	(*Allow Robots to Proceed Into Tool*)
	(*!!!!!This is the final OK to allow Robots Into the Tool Area, So it Better Be Ready!!!!!!!*)
	IF Enable_Motion
		THEN
			IF Load_Robots_Proceed1 AND Load_Robots_WorkingOK1 AND Load_Robots_Clear2 AND Seal_Robots_Clear AND Stud_Robots_Clear AND Turntable_Clear AND Weld_Robots_Clear AND Unload_Robots_Clear
				THEN Robots_Clear_ToProceed:=TRUE;
			ELSIF Load_Robots_Proceed2 AND Load_Robots_WorkingOK2 AND Load_Robots_Clear1 AND Seal_Robots_Clear AND Stud_Robots_Clear AND Turntable_Clear AND Weld_Robots_Clear AND Unload_Robots_Clear
				THEN Robots_Clear_ToProceed:=TRUE;
			ELSIF Seal_Robots_Proceed AND Seal_Robots_WorkingOK AND Load_Robots_Clear AND Stud_Robots_Clear AND Turntable_Clear AND Weld_Robots_Clear AND Unload_Robots_Clear
				THEN Robots_Clear_ToProceed:=TRUE;
			ELSIF Stud_Robots_Proceed AND Stud_Robots_WorkingOK AND Load_Robots_Clear AND Seal_Robots_Clear AND Turntable_Clear AND Weld_Robots_Clear AND Unload_Robots_Clear
				THEN Robots_Clear_ToProceed:=TRUE;
			ELSIF Weld_Robots_Proceed AND Weld_Robots_WorkingOK AND Load_Robots_Clear AND Seal_Robots_Clear AND Stud_Robots_Clear AND Turntable_Clear AND Unload_Robots_Clear
				THEN Robots_Clear_ToProceed:=TRUE;
			ELSIF Unload_Robots_Proceed1 AND Unload_Robots_WorkingOK1 AND Load_Robots_Clear AND Seal_Robots_Clear AND Stud_Robots_Clear AND Turntable_Clear AND Weld_Robots_Clear AND Unload_Robots_Clear2
				THEN Robots_Clear_ToProceed:=TRUE;
			ELSIF Unload_Robots_Proceed2 AND Unload_Robots_WorkingOK2 AND Load_Robots_Clear AND Seal_Robots_Clear AND Stud_Robots_Clear AND Turntable_Clear AND Weld_Robots_Clear AND Unload_Robots_Clear1
				THEN Robots_Clear_ToProceed:=TRUE;
			ELSE Robots_Clear_ToProceed:= FALSE;
			END_IF;
		ELSE Robots_Clear_ToProceed:= FALSE;
	END_IF;

(*+++++++++++++++++++++++++++++++++++++++++++++++ Task Complete Acks ++++++++++++++++++++++++++*)
	(*1st Load Complete Ack*)
	Load_Complete1_Ack:= Load_Robots_Complete1 AND Load_Complete1;

	(*2nd Load Complete Ack*)
	Load_Complete2_Ack:= Load_Robots_Complete2 AND Load_Complete2;

	(*Seal Complete Ack*)
	Seal_Complete_Ack:= Seal_Robots_Complete AND Sealing_Complete;

	(*Stud Complete Ack*)
	Stud_Complete_Ack:= Stud_Robots_Complete AND Stud_Complete;

	(*Sweep Complete ACK*)
	TurnA_Complete_Ack := TurntableA_Complete AND TurntableA_At_Robot;
	TurnB_Complete_Ack := TurntableB_Complete AND TurntableB_At_Robot;

	(*Weld Complete Ack*)
	Weld_Complete_Ack:= Weld_Robots_Complete AND Welding_Complete;

	(*Unload Complete Ack*)
	Unload_Complete1_Ack:= Unload_Robots_Complete1 AND Unload_Complete;

	(*Unload Complete Ack*)
	Unload_Complete2_Ack:= Unload_Robots_Complete2 AND Unload_Complete;






(*end*)
END_ACTION

ACTION Status_and_Faults:



(*^^^^^^^^^^^^^^^^^^^^^^^^^^^^^^^^^^^^^^ General Visualization ^^^^^^^^^^^^^^^^^^^^^^^^^^^^^^^^^^^^*)
	(*For Ready to Load Indicators*)
		(*Flash when tool should be loaded but load is not complete*)
		IF In_Auto AND Tool_At_Home AND NOT Welding_Complete AND All_Robots_Clear AND NOT All_Sensors_On.2
			THEN
				Ready_To_Load:= Pulse_500mS;
				(*Go solid when tool has been loaded properly*)
				(*Go solid when tool is ready to be unloaded*)
		ELSIF In_Auto AND All_Robots_Clear  AND ((Tool_At_Home AND NOT Welding_Complete AND All_Sensors_On.2 AND NOT Enable_Motion)
			OR (Tool_At_Unload.0 AND Welding_Complete AND (Sealing_Complete OR Sealer_Bypass) AND (Stud_Complete OR Stud_Bypass) AND TurntableA_At_Robot AND NOT All_Sensors_Off))
			THEN
				Ready_To_Load:= TRUE;
		ELSE
				Ready_To_Load:= FALSE;
		END_IF;
	(*For Red Stack Light Indicators*)
		Red_Lamp_Req:= PPFaults<>0 OR CLFaulted.0 OR CLFaulted.4 OR (NOT Sealer_Bypass AND MAIN.SL01.Disp1_Volume_NotOK AND (MAIN.R1.Task_ID_Ack=Seal_Fix01)) OR Load_Seq01.Faulted;


	(*Status Banners*)
		(*1 - Check Parts On Sub Check*)
		IF In_Auto AND NOT In_Manual AND NOT Cycle_Complete AND Tool_At_Load.0
			AND NOT Start_Load_Robots1 AND NOT Start_Load_Robots2 AND NOT Start_Seal_Robots AND NOT Start_Stud_Robots AND NOT Start_TurntableA
			AND NOT Start_TurntableB AND NOT Start_Weld_Robots AND NOT Start_Unload_Robots1 AND NOT Start_Unload_Robots2
			THEN
				IF NOT Dry_Cycle AND NOT All_Sensors_On.0
					THEN Status:= 1;
				ELSIF Dry_Cycle AND NOT Load_Complete1
					THEN Status:=1;
				END_IF;
		END_IF;
		(*2 - Sub Check OK*)
		IF In_Auto AND NOT In_Manual AND NOT Cycle_Complete AND Tool_At_Load.1
			AND NOT Start_Load_Robots1 AND NOT Start_Load_Robots2 AND NOT Start_Seal_Robots AND NOT Start_Stud_Robots AND NOT Start_TurntableA
			AND NOT Start_TurntableB AND NOT Start_Weld_Robots AND NOT Start_Unload_Robots1 AND NOT Start_Unload_Robots2
			THEN
				IF NOT Dry_Cycle AND NOT All_Sensors_On.1
					THEN Status:= 2;
				ELSIF Dry_Cycle AND NOT Load_Complete2
					THEN Status:=2;
				END_IF;
		END_IF;
		(*3 - Load Main Part*)
		IF In_Auto AND NOT In_Manual AND NOT Cycle_Complete AND Tool_At_Home
			AND NOT Start_Load_Robots1 AND NOT Start_Load_Robots2 AND NOT Start_Seal_Robots AND NOT Start_Stud_Robots AND NOT Start_TurntableA
			AND NOT Start_TurntableB AND NOT Start_Weld_Robots AND NOT Start_Unload_Robots1 AND NOT Start_Unload_Robots2
			THEN
				IF NOT Dry_Cycle AND NOT All_Sensors_On.2
					THEN Status:= 3;
				ELSIF Dry_Cycle AND NOT Load_Complete
					THEN Status:=3;
				END_IF;
		END_IF;
		(*10 - Load Parts Onto Tool*)
		IF In_Auto AND NOT In_Manual AND NOT Cycle_Complete AND Tool_At_Load.0
			AND NOT Start_Load_Robots1 AND NOT Start_Load_Robots2 AND NOT Start_Seal_Robots AND NOT Start_Stud_Robots AND NOT Start_TurntableA
			AND NOT Start_TurntableB AND NOT Start_Weld_Robots AND NOT Start_Unload_Robots1 AND NOT Start_Unload_Robots2
			THEN
				IF NOT Dry_Cycle AND NOT All_Sensors_On.2
					THEN Status:= 10;
				ELSIF Dry_Cycle AND NOT Load_Complete
					THEN Status:=10;
				END_IF;
		END_IF;
		(*11 - Robot(s) Loading*)
		IF ((Start_Load_Robots1 OR  Load_Robots_WorkingOK1) OR (Start_Load_Robots2 OR  Load_Robots_WorkingOK2)) AND In_Auto AND NOT In_Manual
			AND NOT Start_Seal_Robots AND NOT Start_Stud_Robots AND NOT Start_TurntableA
			AND NOT Start_TurntableB AND NOT Start_Weld_Robots AND NOT Start_Unload_Robots1 AND NOT Start_Unload_Robots2
			THEN Status:= 11;
		END_IF;
		(*12 - Parts Loaded OK*)
		IF In_Auto AND NOT In_Manual AND NOT Cycle_Complete
			AND NOT Start_Load_Robots1 AND NOT Start_Load_Robots2 AND NOT Start_Seal_Robots AND NOT Start_Stud_Robots AND NOT Start_TurntableA
			 AND NOT Start_TurntableB AND NOT Start_Weld_Robots AND NOT Start_Unload_Robots1 AND NOT Start_Unload_Robots2
			THEN
				IF (All_Sensors_On.2 AND Tool_At_Load.0) AND NOT Dry_Cycle
					THEN Status:= 12;
				ELSIF Load_Complete
					THEN Status:= 12;
				END_IF;
		END_IF;
		(*19 - Robot(s) Stud*)
		IF (Start_Stud_Robots OR Stud_Robots_WorkingOK) AND In_Auto AND NOT In_Manual
			AND NOT Start_Load_Robots1 AND NOT Start_Load_Robots2 AND NOT Start_Weld_Robots AND NOT Start_Seal_Robots AND NOT Start_TurntableA
			 AND NOT Start_TurntableB AND NOT Start_Unload_Robots1 AND NOT Start_Unload_Robots2
			THEN Status:= 19;
		END_IF;
		(*20 - Robot(s) Sealing*)
		IF (Start_Seal_Robots OR Seal_Robots_WorkingOK) AND In_Auto AND NOT In_Manual
			AND NOT Start_Load_Robots1 AND NOT Start_Load_Robots2 AND NOT Start_Weld_Robots AND NOT Start_Stud_Robots AND NOT Start_TurntableA
			 AND NOT Start_TurntableB AND NOT Start_Unload_Robots1 AND NOT Start_Unload_Robots2
			THEN Status:= 20;
		END_IF;
		(*21 - Robot(s) Welding*)
		IF (Start_Weld_Robots OR Weld_Robots_WorkingOK) AND In_Auto AND NOT In_Manual
			AND NOT Start_Load_Robots1 AND NOT Start_Load_Robots2 AND NOT Start_Seal_Robots AND NOT Start_Stud_Robots AND NOT Start_TurntableA
			 AND NOT Start_TurntableB AND NOT Start_Unload_Robots1 AND NOT Start_Unload_Robots2
			THEN Status:= 21;
		END_IF;
		(*22 - Welding Complete / Ready for Unload*)
		IF In_Auto AND NOT In_Manual AND NOT Cycle_Complete AND Welding_Complete
			AND NOT Start_Load_Robots1 AND NOT Start_Load_Robots2 AND NOT Start_Seal_Robots AND NOT Start_Stud_Robots AND NOT Start_TurntableA
			AND NOT Start_TurntableB AND NOT Start_Weld_Robots AND NOT Start_Unload_Robots1 AND NOT Start_Unload_Robots2
			THEN Status:= 22;
		END_IF;
		(*26 - Ready for Rotate*)
		IF (Start_TurntableA OR Start_TurntableB) AND In_Auto AND NOT In_Manual
			AND NOT Start_Load_Robots1 AND NOT Start_Load_Robots2 AND NOT Start_Seal_Robots AND NOT Start_Stud_Robots
			AND NOT Start_Weld_Robots AND NOT Start_Unload_Robots1 AND NOT Start_Unload_Robots2
			THEN Status := 26;
		END_IF;
		(*31 - Robot(s) Unloading*)
		IF (Start_Unload_Robots1 OR Unload_Robots_WorkingOK1 OR Start_Unload_Robots2 OR Unload_Robots_WorkingOK2) AND In_Auto AND NOT In_Manual
			AND NOT Start_Load_Robots1 AND NOT Start_Load_Robots2 AND NOT Start_Seal_Robots AND NOT Start_Stud_Robots AND NOT Start_TurntableA
			AND NOT Start_TurntableB AND NOT Start_Weld_Robots
			THEN Status:= 31;
		END_IF;
		(*32 - Unload Complete*)
		IF In_Auto AND NOT In_Manual AND NOT Cycle_Complete AND Unload_Complete
			AND NOT Start_Load_Robots1 AND NOT Start_Load_Robots2 AND NOT Start_Seal_Robots AND NOT Start_Stud_Robots AND NOT Start_TurntableA
			AND NOT Start_TurntableB AND NOT Start_Weld_Robots AND NOT Start_Unload_Robots1 AND NOT Start_Unload_Robots2
			THEN Status:= 32;
		END_IF;
		(*42 - Cycle Complete*)
		IF In_Auto AND NOT In_Manual AND Cycle_Complete AND All_Sensors_Off
			THEN Status:= 42;
		END_IF;
		(*50 - In Manual*)
		IF In_Manual
			THEN Status:= 50;
		END_IF;
		(*51 - Clamp Fault*)
		IF (CLFaults1>0 OR CLFaults2>0 OR CLFaults3>0 OR CLFaults4>0) AND In_Auto AND NOT In_Manual
			THEN Status:= 51;
		END_IF;
		(*52 - Part Present Sensor Fault*)
		IF PPFaults>0 AND In_Auto AND NOT In_Manual
			THEN Status:= 52;
		END_IF;
		(*53 - Nut Checks Failed Call QA*)
		IF QAChecks_Failed AND In_Auto AND NOT In_Manual
			THEN Status:= 53;
		END_IF;
		(*54 - Sealer Failed Call QA*)
		IF NOT Sealer_Bypass AND (MAIN.SL01.Disp1_Volume_NotOK AND (MAIN.R1.Task_ID_Ack=Seal_Fix01)) AND In_Auto AND NOT In_Manual
			THEN Status:= 54;
		END_IF;
		(*55 - Load Sequence Fault Call QA*)
		IF Load_Seq01.Faulted AND In_Auto AND NOT In_Manual
			THEN Status:= 55;
		END_IF;



(*$$$$$$$$$$$$$$$$$$$$$$$$$$$$$$$$$$$$$$$$$$$$$$$$$$$ Faults $$$$$$$$$$$$$$$$$$$$$$$$$$$$$$$$$$$$$$$$$$$$$$$$$$$$$$$*)

	(*Clamp/Cylider Faults Group 1*)
		IF CLFaults1>0
			THEN CLFaulted.1:=TRUE;
		ELSE
			CLFaulted.1:=FALSE;
		END_IF;
	(*Clamp/Cylider Faults Group 2*)
		IF CLFaults2>0
			THEN CLFaulted.2:=TRUE;
		ELSE
			CLFaulted.2:=FALSE;
		END_IF;
	(*Clamp/Cylider Faults Group 3*)
		IF CLFaults3>0
			THEN CLFaulted.3:=TRUE;
		ELSE
			CLFaulted.3:=FALSE;
		END_IF;
	(*Clamp/Cylinder Faults Group 4 - Reserved Flag for QA Check Motion Faults*)
		IF CLFaults4>0
			THEN CLFaulted.4:=TRUE;
		ELSE
			CLFaulted.4:=FALSE;
		END_IF;
	(*Bit 0 is designated as ANY Clamp Group Faulted*)
	IF CLFaulted.1 OR CLFaulted.2 OR CLFaulted.3
		THEN CLFaulted.0:= TRUE;
	ELSE CLFaulted.0 := FALSE;
	END_IF;

	(*Part Present Sensor Faults*)
		IF (PPFaults>0) OR (PPFaults1>0) OR (PPFaults2>0)
			THEN PPFaulted.0:=TRUE;
		ELSE
			PPFaulted.0:=FALSE;
		END_IF;
























(*end*)
END_ACTION

ACTION Task_Fix_Model_IDs:


	(*Develop Task IDs - See Global Variable, "TaskID_Record"*)

	IF (Start_Load_Robots1 OR Start_Load_Robots2) AND Enable_Motion
		THEN Task_ID:= Dropoff_Fix04;
	ELSIF Start_Seal_Robots AND Enable_Motion
		THEN Task_ID:= Seal_Fix04;
	ELSIF Start_Stud_Robots AND Enable_Motion
		THEN Task_ID:= Stud_Fix04;
	ELSIF Start_Weld_Robots AND Enable_Motion
		THEN Task_ID:= Weld_Fix04;
	ELSIF Start_TurnTableB AND Enable_Motion
		THEN Task_ID:= Sweep_Fix04;
	ELSIF (Start_Unload_Robots1 OR Start_Unload_Robots2) AND Enable_Motion
		THEN Task_ID:= Pickup_Fix04;
	ELSE Task_ID:= 0;
	END_IF;

	(*Develop Fixture ID*)
	Fix_ID:= N00.ID;					(*In Future Map Beckhoff Dip Switch Data From IP67 Block to Here*)

	(*Develop Model ID*)
	Model_ID:= Discrete_In.ModelData;
END_ACTION

ACTION Tool_States:


(*+++++++++++THIS AREA IS CUSTOM PER INSTALLATION AND WILL HAVE TO BE MODIFIED PER +++++++++++++*)
(*+++++++++++THIS AREA IS CUSTOM PER INSTALLATION AND WILL HAVE TO BE MODIFIED PER +++++++++++++*)

(*
						 MODEL ID MAP
					 -------------------
				Model ID :  Part ID  :   Tooling ID
					1  	 : 	 504     :     42
					2	 :   524     :	   42
					3	 :   543     :	   47
					4	 :   526     :	   46
					5	 :   536     :	   45
					6	 :   550     :	   44
					7	 :   571     :	   43
	
*)
	

	(*Tooling Position at HOME*)
	Tool_At_HOME:= 
				(((Model_ID=1) OR (Model_ID>3 OR (Model_ID=0)))		(*Model 504, 526, 536, 550, 571*)
				AND Clamp1RETD AND Clamp2RETD AND Clamp3RETD AND Clamp4RETD
				AND Clamp5RETD AND Clamp6RETD AND Clamp7RETD AND Clamp8RETD
				AND Clamp9RETD AND Clamp10RETD AND Clamp11RETD AND Clamp12RETD
				AND Clamp13RETD AND Clamp14RETD AND Clamp15RETD AND Clamp16RETD
				AND Clamp17RETD AND Clamp18RETD AND Clamp19RETD AND Clamp20RETD
				AND Clamp21RETD AND Clamp22RETD AND Pin1ADVD AND Pin2ADVD AND Pin3ADVD AND Pin4ADVD 
				AND Pin5RETD AND Pin6RETD AND Pin7ADVD AND Pin8ADVD AND Pin9ADVD AND Pin10ADVD 
				AND Pin11ADVD AND Pin12ADVD AND Pin13ADVD AND Pin14RETD AND Pin15RETD AND Pin16ADVD AND Pin17ADVD 
				AND Pin18ADVD AND Slide1ADVD AND Slide2ADVD AND Slide3RETD AND Slide4RETD AND Slide5RETD AND Slide6RETD
				AND Slide7RETD AND Slide8RETD AND Slide9RETD AND Slide10ADVD AND Slide11RETD AND Slide12RETD
				AND Slide13ADVD AND Slide14ADVD AND Swing1RETD AND Swing2RETD AND Swing3RETD)
			OR
				((Model_ID=2)		(*524*)
				AND Clamp1RETD AND Clamp2RETD AND Clamp3RETD AND Clamp4RETD
				AND Clamp5RETD AND Clamp6RETD AND Clamp7RETD AND Clamp8RETD
				AND Clamp9RETD AND Clamp10RETD AND Clamp11RETD AND Clamp12RETD
				AND Clamp13RETD AND Clamp14RETD AND Clamp15RETD AND Clamp16RETD
				AND Clamp17RETD AND Clamp18RETD AND Clamp19RETD AND Clamp20RETD
				AND Clamp21RETD AND Clamp22RETD AND Pin1ADVD AND Pin2ADVD AND Pin3ADVD AND Pin4ADVD 
				AND Pin5ADVD AND Pin6RETD AND Pin7ADVD AND Pin8ADVD AND Pin9ADVD AND Pin10ADVD 
				AND Pin11ADVD AND Pin12ADVD AND Pin13ADVD AND Pin14RETD AND Pin15ADVD AND Pin16ADVD AND Pin17ADVD 
				AND Pin18ADVD AND Slide1ADVD AND Slide2ADVD AND Slide3RETD AND Slide4RETD AND Slide5RETD AND Slide6RETD
				AND Slide7RETD AND Slide8RETD AND Slide9RETD AND Slide10ADVD AND Slide11RETD AND Slide12RETD
				AND Slide13ADVD AND Slide14ADVD AND Swing1RETD AND Swing2RETD AND Swing3RETD)
			OR
				((Model_ID=3)		(*543*)
				AND Clamp1RETD AND Clamp2RETD AND Clamp3RETD AND Clamp4RETD
				AND Clamp5RETD AND Clamp6RETD AND Clamp7RETD AND Clamp8RETD
				AND Clamp9RETD AND Clamp10RETD AND Clamp11RETD AND Clamp12RETD
				AND Clamp13RETD AND Clamp14RETD AND Clamp15RETD AND Clamp16RETD
				AND Clamp17RETD AND Clamp18RETD AND Clamp19RETD AND Clamp20RETD
				AND Clamp21RETD AND Clamp22RETD AND Pin1ADVD AND Pin2ADVD AND Pin3ADVD AND Pin4ADVD 
				AND Pin5RETD AND Pin6ADVD AND Pin7ADVD AND Pin8ADVD AND Pin9ADVD AND Pin10ADVD 
				AND Pin11ADVD AND Pin12ADVD AND Pin13ADVD AND Pin14ADVD AND Pin15RETD AND Pin16ADVD AND Pin17ADVD 
				AND Pin18ADVD AND Slide1ADVD AND Slide2ADVD AND Slide3RETD AND Slide4RETD AND Slide5RETD AND Slide6RETD
				AND Slide7RETD AND Slide8RETD AND Slide9RETD AND Slide10ADVD AND Slide11RETD AND Slide12RETD
				AND Slide13ADVD AND Slide14ADVD AND Swing1RETD AND Swing2RETD AND Swing3RETD);

	(*Tooling position to load parts*)
	Tool_At_Load.0:=
				(((Model_ID=1) OR (Model_ID>3))		(*Model 504, 526, 536, 550, 571*)
				AND Clamp1RETD AND Clamp2RETD AND Clamp3RETD AND Clamp4RETD
				AND Clamp5RETD AND Clamp6RETD AND Clamp7RETD AND Clamp8RETD
				AND Clamp9RETD AND Clamp10RETD AND Clamp11RETD AND Clamp12RETD
				AND Clamp13RETD AND Clamp14RETD AND Clamp15RETD AND Clamp16RETD
				AND Clamp17RETD AND Clamp18RETD AND Clamp19RETD AND Clamp20RETD
				AND Clamp21RETD AND Clamp22RETD AND Pin1ADVD AND Pin2ADVD AND Pin3ADVD AND Pin4ADVD 
				AND Pin5RETD AND Pin6RETD AND Pin7ADVD AND Pin8ADVD AND Pin9ADVD AND Pin10ADVD 
				AND Pin11ADVD AND Pin12ADVD AND Pin13ADVD AND Pin14RETD AND Pin15RETD AND Pin16ADVD AND Pin17ADVD 
				AND Pin18ADVD AND Slide1ADVD AND Slide2ADVD AND Slide3RETD AND Slide4RETD AND Slide5RETD AND Slide6RETD
				AND Slide7RETD AND Slide8RETD AND Slide9RETD AND Slide10ADVD AND Slide11RETD AND Slide12RETD
				AND Slide13ADVD AND Slide14ADVD AND Swing1RETD AND Swing2RETD AND Swing3RETD)
			OR
				((Model_ID=2)		(*Model 524*)
				AND Clamp1RETD AND Clamp2RETD AND Clamp3RETD AND Clamp4RETD
				AND Clamp5RETD AND Clamp6RETD AND Clamp7RETD AND Clamp8RETD
				AND Clamp9RETD AND Clamp10RETD AND Clamp11RETD AND Clamp12RETD
				AND Clamp13RETD AND Clamp14RETD AND Clamp15RETD AND Clamp16RETD
				AND Clamp17RETD AND Clamp18RETD AND Clamp19RETD AND Clamp20RETD
				AND Clamp21RETD AND Clamp22RETD AND Pin1ADVD AND Pin2ADVD AND Pin3ADVD AND Pin4ADVD 
				AND Pin5ADVD AND Pin6RETD AND Pin7ADVD AND Pin8ADVD AND Pin9ADVD AND Pin10ADVD 
				AND Pin11ADVD AND Pin12ADVD AND Pin13ADVD AND Pin14RETD AND Pin15ADVD AND Pin16ADVD AND Pin17ADVD 
				AND Pin18ADVD AND Slide1ADVD AND Slide2ADVD AND Slide3RETD AND Slide4RETD AND Slide5RETD AND Slide6RETD
				AND Slide7RETD AND Slide8RETD AND Slide9RETD AND Slide10ADVD AND Slide11RETD AND Slide12RETD
				AND Slide13ADVD AND Slide14ADVD AND Swing1RETD AND Swing2RETD AND Swing3RETD)
			OR
				((Model_ID=3)		(*Model 543*)
				AND Clamp1RETD AND Clamp2RETD AND Clamp3RETD AND Clamp4RETD
				AND Clamp5RETD AND Clamp6RETD AND Clamp7RETD AND Clamp8RETD
				AND Clamp9RETD AND Clamp10RETD AND Clamp11RETD AND Clamp12RETD
				AND Clamp13RETD AND Clamp14RETD AND Clamp15RETD AND Clamp16RETD
				AND Clamp17RETD AND Clamp18RETD AND Clamp19RETD AND Clamp20RETD
				AND Clamp21RETD AND Clamp22RETD AND Pin1ADVD AND Pin2ADVD AND Pin3ADVD AND Pin4ADVD 
				AND Pin5RETD AND Pin6ADVD AND Pin7ADVD AND Pin8ADVD AND Pin9ADVD AND Pin10ADVD 
				AND Pin11ADVD AND Pin12ADVD AND Pin13ADVD AND Pin14ADVD AND Pin15RETD AND Pin16ADVD AND Pin17ADVD 
				AND Pin18ADVD AND Slide1ADVD AND Slide2ADVD AND Slide3RETD AND Slide4RETD AND Slide5RETD AND Slide6RETD
				AND Slide7RETD AND Slide8RETD AND Slide9RETD AND Slide10ADVD AND Slide11RETD AND Slide12RETD
				AND Slide13ADVD AND Slide14ADVD AND Swing1RETD AND Swing2RETD AND Swing3RETD);
	
	(*Tooling position on Loading Complete*)	
	Tool_At_Load.1:= 
				(((Model_ID=1) OR (Model_ID>3))		(*Model 504, 526, 536, 550, 571*)
				AND Clamp1ADVD AND Clamp2ADVD AND Clamp3ADVD AND Clamp4ADVD AND Clamp5ADVD AND Clamp5ADVD AND Clamp5ADVD
				AND Clamp6ADVD AND Clamp7ADVD AND Clamp8ADVD AND Clamp9ADVD AND Clamp10ADVD AND Clamp11ADVD AND Clamp12ADVD
				AND Clamp13ADVD AND Clamp14ADVD AND Clamp15ADVD AND Clamp16ADVD AND Clamp17ADVD AND Clamp18ADVD AND Clamp19ADVD
				AND Clamp20ADVD AND Clamp21ADVD AND Clamp22ADVD AND Pin1ADVD AND Pin2ADVD AND Pin3ADVD AND Pin4ADVD AND Pin5RETD
				AND Pin6RETD AND Pin7ADVD AND Pin8ADVD AND Pin9ADVD AND Pin10ADVD AND Pin11ADVD AND Pin12ADVD AND Pin13ADVD
				AND Pin14RETD AND Pin15RETD AND Pin16ADVD AND Pin17ADVD AND Pin18ADVD AND Slide1ADVD AND Slide2ADVD AND Slide3ADVD
				AND Slide4ADVD AND Slide5ADVD AND Slide6ADVD AND Slide7ADVD AND Slide8ADVD AND Slide9ADVD AND Slide10ADVD AND Slide11ADVD
				AND Slide12ADVD AND Slide13ADVD AND Slide14ADVD AND Swing1ADVD AND Swing2ADVD AND Swing3ADVD)
			OR
				((Model_ID=2)		(*Model 524*)
				AND Clamp1ADVD AND Clamp2ADVD AND Clamp3ADVD AND Clamp4ADVD AND Clamp5ADVD AND Clamp5ADVD AND Clamp5ADVD
				AND Clamp6ADVD AND Clamp7ADVD AND Clamp8ADVD AND Clamp9ADVD AND Clamp10ADVD AND Clamp11ADVD AND Clamp12ADVD
				AND Clamp13ADVD AND Clamp14ADVD AND Clamp15ADVD AND Clamp16ADVD AND Clamp17ADVD AND Clamp18ADVD AND Clamp19ADVD
				AND Clamp20ADVD AND Clamp21ADVD AND Clamp22ADVD AND Pin1ADVD AND Pin2ADVD AND Pin3ADVD AND Pin4ADVD AND Pin5ADVD
				AND Pin6RETD AND Pin7ADVD AND Pin8ADVD AND Pin9ADVD AND Pin10ADVD AND Pin11ADVD AND Pin12ADVD AND Pin13ADVD
				AND Pin14RETD AND Pin15ADVD AND Pin16ADVD AND Pin17ADVD AND Pin18ADVD AND Slide1ADVD AND Slide2ADVD AND Slide3ADVD
				AND Slide4ADVD AND Slide5ADVD AND Slide6ADVD AND Slide7ADVD AND Slide8ADVD AND Slide9ADVD AND Slide10ADVD AND Slide11ADVD
				AND Slide12ADVD AND Slide13ADVD AND Slide14ADVD AND Swing1ADVD AND Swing2ADVD AND Swing3ADVD)
			OR
				((Model_ID=3)		(*Model 543*)
				AND Clamp1ADVD AND Clamp2ADVD AND Clamp3ADVD AND Clamp4ADVD AND Clamp5ADVD AND Clamp5ADVD AND Clamp5ADVD
				AND Clamp6ADVD AND Clamp7ADVD AND Clamp8ADVD AND Clamp9ADVD AND Clamp10ADVD AND Clamp11ADVD AND Clamp12ADVD
				AND Clamp13ADVD AND Clamp14ADVD AND Clamp15ADVD AND Clamp16ADVD AND Clamp17ADVD AND Clamp18ADVD AND Clamp19ADVD
				AND Clamp20ADVD AND Clamp21ADVD AND Clamp22ADVD AND Pin1ADVD AND Pin2ADVD AND Pin3ADVD AND Pin4ADVD AND Pin5RETD
				AND Pin6ADVD AND Pin7ADVD AND Pin8ADVD AND Pin9ADVD AND Pin10ADVD AND Pin11ADVD AND Pin12ADVD AND Pin13ADVD
				AND Pin14ADVD AND Pin15RETD AND Pin16ADVD AND Pin17ADVD AND Pin18ADVD AND Slide1ADVD AND Slide2ADVD AND Slide3ADVD
				AND Slide4ADVD AND Slide5ADVD AND Slide6ADVD AND Slide7ADVD AND Slide8ADVD AND Slide9ADVD AND Slide10ADVD AND Slide11ADVD
				AND Slide12ADVD AND Slide13ADVD AND Slide14ADVD AND Swing1ADVD AND Swing2ADVD AND Swing3ADVD);
	Tool_At_Load.2:= FALSE;
	Tool_At_Load.3:= FALSE;
	Tool_At_Load.4:= FALSE;


	Tool_At_Seal.0:= FALSE;
	Tool_At_Seal.1:= FALSE;
	Tool_At_Seal.2:= FALSE;
	Tool_At_Seal.3:= FALSE;
	Tool_At_Seal.4:= FALSE;


	Tool_At_Stud.0:= FALSE;
	Tool_At_Stud.1:= FALSE;
	Tool_At_Stud.2:= FALSE;
	Tool_At_Stud.3:= FALSE;
	Tool_At_Stud.4:= FALSE;

	(*Tooling position for ready to rotate*)
	Tool_At_Rotate.0:= 
				(((Model_ID=1) OR (Model_ID>3))		(*Model 504, 526, 536, 550, 571*)
				AND Clamp1ADVD AND Clamp2ADVD AND Clamp3ADVD AND Clamp4ADVD AND Clamp5ADVD AND Clamp5ADVD AND Clamp5ADVD
				AND Clamp6ADVD AND Clamp7ADVD AND Clamp8ADVD AND Clamp9ADVD AND Clamp10ADVD AND Clamp11ADVD AND Clamp12ADVD
				AND Clamp13ADVD AND Clamp14ADVD AND Clamp15ADVD AND Clamp16ADVD AND Clamp17ADVD AND Clamp18ADVD AND Clamp19ADVD
				AND Clamp20ADVD AND Clamp21ADVD AND Clamp22ADVD AND Pin1ADVD AND Pin2ADVD AND Pin3ADVD AND Pin4ADVD AND Pin5RETD
				AND Pin6RETD AND Pin7ADVD AND Pin8ADVD AND Pin9ADVD AND Pin10ADVD AND Pin11ADVD AND Pin12ADVD AND Pin13ADVD
				AND Pin14RETD AND Pin15RETD AND Pin16ADVD AND Pin17ADVD AND Pin18ADVD AND Slide1ADVD AND Slide2ADVD AND Slide3ADVD
				AND Slide4ADVD AND Slide5ADVD AND Slide6ADVD AND Slide7ADVD AND Slide8ADVD AND Slide9ADVD AND Slide10ADVD AND Slide11ADVD
				AND Slide12ADVD AND Slide13ADVD AND Slide14ADVD AND Swing1ADVD AND Swing2ADVD AND Swing3ADVD)
			OR
				((Model_ID=2)		(*Model 524*)
				AND Clamp1ADVD AND Clamp2ADVD AND Clamp3ADVD AND Clamp4ADVD AND Clamp5ADVD AND Clamp5ADVD AND Clamp5ADVD
				AND Clamp6ADVD AND Clamp7ADVD AND Clamp8ADVD AND Clamp9ADVD AND Clamp10ADVD AND Clamp11ADVD AND Clamp12ADVD
				AND Clamp13ADVD AND Clamp14ADVD AND Clamp15ADVD AND Clamp16ADVD AND Clamp17ADVD AND Clamp18ADVD AND Clamp19ADVD
				AND Clamp20ADVD AND Clamp21ADVD AND Clamp22ADVD AND Pin1ADVD AND Pin2ADVD AND Pin3ADVD AND Pin4ADVD AND Pin5ADVD
				AND Pin6RETD AND Pin7ADVD AND Pin8ADVD AND Pin9ADVD AND Pin10ADVD AND Pin11ADVD AND Pin12ADVD AND Pin13ADVD
				AND Pin14RETD AND Pin15ADVD AND Pin16ADVD AND Pin17ADVD AND Pin18ADVD AND Slide1ADVD AND Slide2ADVD AND Slide3ADVD
				AND Slide4ADVD AND Slide5ADVD AND Slide6ADVD AND Slide7ADVD AND Slide8ADVD AND Slide9ADVD AND Slide10ADVD AND Slide11ADVD
				AND Slide12ADVD AND Slide13ADVD AND Slide14ADVD AND Swing1ADVD AND Swing2ADVD AND Swing3ADVD)
			OR
				((Model_ID=3)		(*Model 543*)
				AND Clamp1ADVD AND Clamp2ADVD AND Clamp3ADVD AND Clamp4ADVD AND Clamp5ADVD AND Clamp5ADVD AND Clamp5ADVD
				AND Clamp6ADVD AND Clamp7ADVD AND Clamp8ADVD AND Clamp9ADVD AND Clamp10ADVD AND Clamp11ADVD AND Clamp12ADVD
				AND Clamp13ADVD AND Clamp14ADVD AND Clamp15ADVD AND Clamp16ADVD AND Clamp17ADVD AND Clamp18ADVD AND Clamp19ADVD
				AND Clamp20ADVD AND Clamp21ADVD AND Clamp22ADVD AND Pin1ADVD AND Pin2ADVD AND Pin3ADVD AND Pin4ADVD AND Pin5RETD
				AND Pin6ADVD AND Pin7ADVD AND Pin8ADVD AND Pin9ADVD AND Pin10ADVD AND Pin11ADVD AND Pin12ADVD AND Pin13ADVD
				AND Pin14ADVD AND Pin15RETD AND Pin16ADVD AND Pin17ADVD AND Pin18ADVD AND Slide1ADVD AND Slide2ADVD AND Slide3ADVD
				AND Slide4ADVD AND Slide5ADVD AND Slide6ADVD AND Slide7ADVD AND Slide8ADVD AND Slide9ADVD AND Slide10ADVD AND Slide11ADVD
				AND Slide12ADVD AND Slide13ADVD AND Slide14ADVD AND Swing1ADVD AND Swing2ADVD AND Swing3ADVD);
				
	Tool_At_Rotate.1:= FALSE;
	Tool_At_Rotate.2:= FALSE;
	Tool_At_Rotate.3:= FALSE;
	Tool_At_Rotate.4:= FALSE;

	(*Tooling position for welding*)
	Tool_At_Weld.0:= 
				(((Model_ID=1) OR (Model_ID>3))		(*Model 504, 526, 536, 550, 571*)
				AND Clamp1ADVD AND Clamp2ADVD AND Clamp3ADVD AND Clamp4ADVD AND Clamp5ADVD AND Clamp5ADVD AND Clamp5ADVD
				AND Clamp6ADVD AND Clamp7ADVD AND Clamp8ADVD AND Clamp9ADVD AND Clamp10ADVD AND Clamp11ADVD AND Clamp12ADVD
				AND Clamp13ADVD AND Clamp14ADVD AND Clamp15ADVD AND Clamp16ADVD AND Clamp17ADVD AND Clamp18ADVD AND Clamp19ADVD
				AND Clamp20ADVD AND Clamp21ADVD AND Clamp22ADVD AND Pin1ADVD AND Pin2ADVD AND Pin3ADVD AND Pin4ADVD AND Pin5RETD
				AND Pin6RETD AND Pin7ADVD AND Pin8ADVD AND Pin9ADVD AND Pin10ADVD AND Pin11ADVD AND Pin12ADVD AND Pin13ADVD
				AND Pin14RETD AND Pin15RETD AND Pin16ADVD AND Pin17ADVD AND Pin18ADVD AND Slide1ADVD AND Slide2ADVD AND Slide3ADVD
				AND Slide4ADVD AND Slide5ADVD AND Slide6ADVD AND Slide7ADVD AND Slide8ADVD AND Slide9ADVD AND Slide10ADVD AND Slide11ADVD
				AND Slide12ADVD AND Slide13ADVD AND Slide14ADVD AND Swing1ADVD AND Swing2ADVD AND Swing3ADVD)
			OR
				((Model_ID=2)		(*Model 524*)
				AND Clamp1ADVD AND Clamp2ADVD AND Clamp3ADVD AND Clamp4ADVD AND Clamp5ADVD AND Clamp5ADVD AND Clamp5ADVD
				AND Clamp6ADVD AND Clamp7ADVD AND Clamp8ADVD AND Clamp9ADVD AND Clamp10ADVD AND Clamp11ADVD AND Clamp12ADVD
				AND Clamp13ADVD AND Clamp14ADVD AND Clamp15ADVD AND Clamp16ADVD AND Clamp17ADVD AND Clamp18ADVD AND Clamp19ADVD
				AND Clamp20ADVD AND Clamp21ADVD AND Clamp22ADVD AND Pin1ADVD AND Pin2ADVD AND Pin3ADVD AND Pin4ADVD AND Pin5ADVD
				AND Pin6RETD AND Pin7ADVD AND Pin8ADVD AND Pin9ADVD AND Pin10ADVD AND Pin11ADVD AND Pin12ADVD AND Pin13ADVD
				AND Pin14RETD AND Pin15ADVD AND Pin16ADVD AND Pin17ADVD AND Pin18ADVD AND Slide1ADVD AND Slide2ADVD AND Slide3ADVD
				AND Slide4ADVD AND Slide5ADVD AND Slide6ADVD AND Slide7ADVD AND Slide8ADVD AND Slide9ADVD AND Slide10ADVD AND Slide11ADVD
				AND Slide12ADVD AND Slide13ADVD AND Slide14ADVD AND Swing1ADVD AND Swing2ADVD AND Swing3ADVD)
			OR
				((Model_ID=3)		(*Model 543*)
				AND Clamp1ADVD AND Clamp2ADVD AND Clamp3ADVD AND Clamp4ADVD AND Clamp5ADVD AND Clamp5ADVD AND Clamp5ADVD
				AND Clamp6ADVD AND Clamp7ADVD AND Clamp8ADVD AND Clamp9ADVD AND Clamp10ADVD AND Clamp11ADVD AND Clamp12ADVD
				AND Clamp13ADVD AND Clamp14ADVD AND Clamp15ADVD AND Clamp16ADVD AND Clamp17ADVD AND Clamp18ADVD AND Clamp19ADVD
				AND Clamp20ADVD AND Clamp21ADVD AND Clamp22ADVD AND Pin1ADVD AND Pin2ADVD AND Pin3ADVD AND Pin4ADVD AND Pin5RETD
				AND Pin6ADVD AND Pin7ADVD AND Pin8ADVD AND Pin9ADVD AND Pin10ADVD AND Pin11ADVD AND Pin12ADVD AND Pin13ADVD
				AND Pin14ADVD AND Pin15RETD AND Pin16ADVD AND Pin17ADVD AND Pin18ADVD AND Slide1ADVD AND Slide2ADVD AND Slide3ADVD
				AND Slide4ADVD AND Slide5ADVD AND Slide6ADVD AND Slide7ADVD AND Slide8ADVD AND Slide9ADVD AND Slide10ADVD AND Slide11ADVD
				AND Slide12ADVD AND Slide13ADVD AND Slide14ADVD AND Swing1ADVD AND Swing2ADVD AND Swing3ADVD);
	Tool_At_Weld.1:= FALSE;
	Tool_At_Weld.2:= FALSE;
	Tool_At_Weld.3:= FALSE;
	Tool_At_Weld.4:= FALSE;

	(*Tooling position for unload*)
	Tool_At_Unload.0:=Clamp1RETD AND Clamp2RETD AND Clamp3RETD AND Clamp4RETD
				AND Clamp5RETD AND Clamp6RETD AND Clamp7RETD AND Clamp8RETD
				AND Clamp9RETD AND Clamp10RETD AND Clamp11RETD AND Clamp12RETD
				AND Clamp13RETD AND Clamp14RETD AND Clamp15RETD AND Clamp16RETD
				AND Clamp17RETD AND Clamp18RETD AND Clamp19RETD AND Clamp20RETD
				AND Clamp21RETD AND Clamp22RETD AND Pin1RETD AND Pin2RETD AND Pin3RETD AND Pin4RETD AND Pin5RETD
				AND Pin6RETD AND Pin7RETD AND Pin8RETD AND Pin9RETD AND Pin10RETD AND Pin11RETD AND Pin12RETD 
				AND Pin13RETD AND Pin14RETD AND Pin15RETD AND Pin16RETD AND Pin17RETD AND Pin18RETD
				AND Slide1RETD AND Slide2RETD AND Slide3RETD AND Slide4RETD AND Slide5RETD AND Slide6RETD
				AND Slide7RETD AND Slide8RETD AND Slide9RETD AND Slide10RETD AND Slide11RETD AND Slide12RETD
				AND Slide13RETD AND Slide14RETD AND Swing1RETD AND Swing2RETD AND Swing3RETD;
	Tool_At_Unload.1:=FALSE;
	Tool_At_Unload.2:= FALSE;
	Tool_At_Unload.3:= FALSE;
	Tool_At_Unload.4:= FALSE;







































(*end*)
END_ACTION

ACTION Tool_VBSeq_Repos:
(*+++++++++++THIS AREA IS CUSTOM PER INSTALLATION AND WILL HAVE TO BE MODIFIED PER +++++++++++++*)
(*+++++++++++THIS AREA IS CUSTOM PER INSTALLATION AND WILL HAVE TO BE MODIFIED PER +++++++++++++*)


(*!!!!!!!!!!!!!!!!!!!!!!!!!!!!!!!!!!!!!!!!!! Tool Motion Control !!!!!!!!!!!!!!!!!!!!!!!!!!!!!!!*)

(*----------------------------------------- Clamp / Unclamp Steps -------------------------------*)

(*$$$$$$$$$$$$$$$$$$$$$$$$$$$$$$$$$$ Develop Clamp and Unclamp Interlocks $$$$$$$$$$$$$$$$$$$$$$*)
(* Note: This is one method to create valve bank commands for clamp and unclamp sequencing
you are welcome to use the direct method as well*)


	(*---------------------------------------------------------Start Clamp Sequence---------------------------------------------------------*)
	
	(*First Stage Clamping*)		(*V8, V10 ADV, IF Model 2 then V2 ADV, IF Model 3 then V5 ADV*)
	Clamp_Step.0:= Auto_Run AND NOT Welding_Complete OR (Cycle_Complete AND NOT Tool_At_Home AND All_Sensors_Off);
	
	
	(*Second Stage Clamping*)		(*V7, V9, V11 ADV, IF Model 2 then V1 ADV, IF Model 3 V4 ADV*)
	
	(*Model 504, 526, 536, 550, 571*)
	IF (Model_ID=1) OR (Model_ID>3) THEN		
				Clamp_Step.1:=  Clamp_Step.0 AND Load_Complete AND NOT Cycle_Complete AND
								(*V8*)
								(Pin1ADVD AND Pin2ADVD AND Pin3ADVD AND Pin4ADVD AND Pin7ADVD 
								AND Pin9ADVD AND Pin16ADVD AND Pin17ADVD AND Pin18ADVD AND Slide10ADVD)
								(*V10*)
								AND (Pin8ADVD AND Pin10ADVD AND Pin11ADVD AND Pin12ADVD AND Pin13ADVD 
								AND Slide1ADVD AND Slide2ADVD AND Slide13ADVD AND Slide14ADVD);
		(*Model 524*)						
		ELSIF (Model_ID=2) THEN					
				Clamp_Step.1:=  Clamp_Step.0 AND Load_Complete AND NOT Cycle_Complete AND 
								(*V2*)
								(Pin5ADVD AND Pin15ADVD)
								(*V8*)
								AND (Pin1ADVD AND Pin2ADVD AND Pin3ADVD AND Pin4ADVD AND Pin7ADVD 
								AND Pin9ADVD AND Pin16ADVD AND Pin17ADVD AND Pin18ADVD AND Slide10ADVD)
								(*V10*)
								AND (Pin8ADVD AND Pin10ADVD AND Pin11ADVD AND Pin12ADVD AND Pin13ADVD 
								AND Slide1ADVD AND Slide2ADVD AND Slide13ADVD AND Slide14ADVD);
		(*Model 543*)			
		ELSIF (Model_ID=3) THEN					
				Clamp_Step.1:=  Clamp_Step.0 AND Load_Complete AND NOT Cycle_Complete AND 
								(*V5*)
								(Pin6ADVD AND Pin14ADVD)
								(*V8*)
								AND (Pin1ADVD AND Pin2ADVD AND Pin3ADVD AND Pin4ADVD AND Pin7ADVD 
								AND Pin9ADVD AND Pin16ADVD AND Pin17ADVD AND Pin18ADVD AND Slide10ADVD)
								(*V10*)
								AND (Pin8ADVD AND Pin10ADVD AND Pin11ADVD AND Pin12ADVD AND Pin13ADVD 
								AND Slide1ADVD AND Slide2ADVD AND Slide13ADVD AND Slide14ADVD);						
	END_IF

	
	(*Third Stage Clamping*)		(*V13 ADV*)
	
	(*Model 504, 526, 536, 550, 571*)
	IF (Model_ID=1) OR (Model_ID>3) THEN
				Clamp_Step.2:= 	Clamp_Step.1 AND 
								(*V7*)
								(Clamp3ADVD AND Clamp18ADVD)
								(*V9*)
								AND (Clamp1ADVD AND Clamp2ADVD AND Clamp4ADVD AND Clamp5ADVD AND Clamp10ADVD 
								AND Clamp14ADVD AND Clamp21ADVD AND Clamp22ADVD)
								(*V11*)
								AND (Clamp9ADVD AND Clamp12ADVD AND Clamp13ADVD AND Clamp16ADVD);

		ELSIF (Model_ID=2) THEN
				Clamp_Step.2:= 	Clamp_Step.1 AND 
								(*V7*)
								(Clamp3ADVD AND Clamp18ADVD)
								(*V9*)
								AND (Clamp1ADVD AND Clamp2ADVD AND Clamp4ADVD AND Clamp5ADVD AND Clamp10ADVD 
								AND Clamp14ADVD AND Clamp21ADVD AND Clamp22ADVD)
								(*V11*)
								AND (Clamp9ADVD AND Clamp12ADVD AND Clamp13ADVD AND Clamp16ADVD)
								(*V1*)
								AND (Clamp6ADVD AND Clamp20ADVD);
		ELSIF (Model_ID=3) THEN
				Clamp_Step.2:= 	Clamp_Step.1 AND 
								(*V7*)
								(Clamp3ADVD AND Clamp18ADVD)
								(*V9*)
								AND (Clamp1ADVD AND Clamp2ADVD AND Clamp4ADVD AND Clamp5ADVD AND Clamp10ADVD 
								AND Clamp14ADVD AND Clamp21ADVD AND Clamp22ADVD)
								(*V11*)
								AND (Clamp9ADVD AND Clamp12ADVD AND Clamp13ADVD AND Clamp16ADVD)
								(*V4*)
								AND (Clamp8ADVD AND Clamp19ADVD);
	END_IF


	(*Forth Stage Clamping*)		(*V12 ADV, IF Model 2 V3 ADV, IF Model 3 V6 ADV*)
	
	Clamp_Step.3:= Clamp_Step.2 AND 
					(*V13*)
					(Clamp7ADVD AND Clamp11ADVD AND Clamp15ADVD AND Clamp17ADVD);




	(*---------------------------------------------------------Start Unclamp Sequence---------------------------------------------------------*)

	(*First Stage Unclamping*)		(*V7, V9, V11 RET, IF Model 2 V1 RET, IF Model 3 V4 RET*)

	Unclamp_Step.0:= (Welding_Complete AND TurnTableA_At_Robot);


	(*Second Stage Unclamping*)		(*V8, V10 RET, IF Model 2 V2 RET, IF Model 3 V5 RET*)
	(*Model 504, 526, 536, 550, 571*)
	IF (Model_ID=1) OR (Model_ID>3) THEN
			Unclamp_Step.1:= Unclamp_Step.0 AND 
								(*V7*)
								(Clamp3RETD AND Clamp18RETD)
								(*V9*)
								AND (Clamp1RETD AND Clamp2RETD AND Clamp4RETD AND Clamp5RETD AND Clamp10RETD AND Clamp14RETD AND Clamp21RETD AND Clamp22RETD)
								(*V11*)
								AND (Clamp9RETD AND Clamp12RETD AND Clamp13RETD AND Clamp16RETD);
		(*Model 524*)							
		ELSIF (Model_ID=2) THEN
				Unclamp_Step.1:= Unclamp_Step.0 AND 
									(*V7*)
									(Clamp3RETD AND Clamp18RETD)
									(*V9*)
									AND (Clamp1RETD AND Clamp2RETD AND Clamp4RETD AND Clamp5RETD AND Clamp10RETD AND Clamp14RETD AND Clamp21RETD AND Clamp22RETD)
									(*V11*)
									AND (Clamp9RETD AND Clamp12RETD AND Clamp13RETD AND Clamp16RETD)
									(*V1*)
									AND (Clamp6RETD AND Clamp20RETD);
		(*Model 543*)
		ELSIF (Model_ID=3) THEN							
				Unclamp_Step.1:= Unclamp_Step.0 AND 
									(*V7*)
									(Clamp3RETD AND Clamp18RETD)
									(*V9*)
									AND (Clamp1RETD AND Clamp2RETD AND Clamp4RETD AND Clamp5RETD AND Clamp10RETD AND Clamp14RETD AND Clamp21RETD AND Clamp22RETD)
									(*V11*)
									AND (Clamp9RETD AND Clamp12RETD AND Clamp13RETD AND Clamp16RETD)
									(*V4*)
									AND (Clamp8RETD AND Clamp19RETD);
	END_IF

	
	(*Third Stage Unclamping*)		(*V12 RET, IF Model 2 V3 RET, IF Model 3 V6 RET*)
	(*Model 504, 526, 536, 550, 571*)
	IF (Model_ID=1) OR (Model_ID>3) THEN
			Unclamp_Step.2:= Unclamp_Step.1 AND 
						(*V8*)
						(Pin1RETD AND Pin2RETD AND Pin3RETD AND Pin4RETD AND Pin7RETD AND Pin9RETD AND Pin16RETD AND Pin17RETD AND Pin18RETD AND Slide10RETD)
						(*V10*)
						AND (Pin8RETD AND Pin10RETD AND Pin11RETD AND Pin12RETD AND Pin13RETD AND Slide1RETD AND Slide2RETD AND Slide13RETD AND Slide14RETD);
		(*Model 524*)
		ELSIF (Model_ID=2) THEN
				Unclamp_Step.2:= Unclamp_Step.1 AND 
							(*V8*)
							(Pin1RETD AND Pin2RETD AND Pin3RETD AND Pin4RETD AND Pin7RETD AND Pin9RETD AND Pin16RETD AND Pin17RETD AND Pin18RETD AND Slide10RETD)
							(*V10*)
							AND (Pin8RETD AND Pin10RETD AND Pin11RETD AND Pin12RETD AND Pin13RETD AND Slide1RETD AND Slide2RETD AND Slide13RETD AND Slide14RETD)
							(*V2*)
							AND (Pin5RETD AND Pin15RETD);
		(*Model 543*)
		ELSIF (Model_ID=3) THEN
				Unclamp_Step.2:= Unclamp_Step.1 AND 
							(*V8*)
							(Pin1RETD AND Pin2RETD AND Pin3RETD AND Pin4RETD AND Pin7RETD AND Pin9RETD AND Pin16RETD AND Pin17RETD AND Pin18RETD AND Slide10RETD)
							(*V10*)
							AND (Pin8RETD AND Pin10RETD AND Pin11RETD AND Pin12RETD AND Pin13RETD AND Slide1RETD AND Slide2RETD AND Slide13RETD AND Slide14RETD)
							(*V5*)
							AND (Pin6RETD AND Pin14RETD);
	
	END_IF

	(*Fourth Stage Unclamping*)		(*V13 RET*)
	(*Model 504, 526, 536, 550, 571*)
	IF (Model_ID=1) OR (Model_ID>3) THEN
				Unclamp_Step.3:= Unclamp_Step.2 AND 
							(*V12*)
							(Slide3RETD AND Slide5RETD AND Slide6RETD AND Slide7RETD AND Slide8RETD AND Slide9RETD AND Slide12RETD AND Swing2RETD);

		ELSIF (Model_ID=2) THEN
				Unclamp_Step.3:= Unclamp_Step.2 AND 
							(*V12*)
							(Slide3RETD AND Slide5RETD AND Slide6RETD AND Slide7RETD AND Slide8RETD AND Slide9RETD AND Slide12RETD AND Swing2RETD)
							(*V3*)
							AND (Slide4RETD AND Slide11RETD);
							
							
		ELSIF (Model_ID=3) THEN
				Unclamp_Step.3:= Unclamp_Step.2 AND 
							(*V12*)
							(Slide3RETD AND Slide5RETD AND Slide6RETD AND Slide7RETD AND Slide8RETD AND Slide9RETD AND Slide12RETD AND Swing2RETD)
							(*V6*)
							AND (Swing1RETD AND Swing3RETD);
							
	END_IF							


(*------------------------------------------- Repositions --------------------------------------*)

	(*Reposition Request#1*)
	IF FALSE
		THEN
			Repo_Reqs.0:= TRUE;
	END_IF;

	(*Reposition Request#2*)
	IF FALSE
		THEN
			Repo_Reqs.1:= TRUE;
	END_IF;

	(*Reposition Request#3*)
	IF FALSE
		THEN
			Repo_Reqs.2:= TRUE;
	END_IF;

	(*Reposition Request#4*)
	IF FALSE
		THEN
			Repo_Reqs.3:= TRUE;
	END_IF;

	(*Reposition Request#5*)
	IF FALSE
		THEN
			Repo_Reqs.4:= TRUE;
	END_IF;

	(*Reposition Request#6*)
	IF FALSE
		THEN
			Repo_Reqs.5:= TRUE;
	END_IF;

	(*Reposition Request#7*)
	IF FALSE
		THEN
			Repo_Reqs.6:= TRUE;
	END_IF;

	(*Reposition Request#8*)
	IF FALSE
		THEN
			Repo_Reqs.7:= TRUE;
	END_IF;

	(*Reset All Reposition Acks At the End Of Cycle*)
	IF Cycle_Complete
		THEN
			Repo_Reqs:= 0;
	END_IF;

(*------------------------- Reposition Acks ---------------------*)
	Repo_Ack.0:= Repo_Reqs.0 AND FALSE;
	Repo_Ack.1:= Repo_Reqs.1 AND FALSE;
	Repo_Ack.2:= Repo_Reqs.2 AND FALSE;
	Repo_Ack.3:= Repo_Reqs.3 AND FALSE;
	Repo_Ack.4:= Repo_Reqs.4 AND FALSE;
	Repo_Ack.5:= Repo_Reqs.5 AND FALSE;
	Repo_Ack.6:= Repo_Reqs.6 AND FALSE;
	Repo_Ack.7:= Repo_Reqs.7 AND FALSE;
END_ACTION

ACTION ValveBank1:


(*+++++++++++THIS AREA IS CUSTOM PER INSTALLATION AND WILL HAVE TO BE MODIFIED PER +++++++++++++*)
(*+++++++++++THIS AREA IS CUSTOM PER INSTALLATION AND WILL HAVE TO BE MODIFIED PER +++++++++++++*)
(*+++++++++++THIS AREA IS CUSTOM PER INSTALLATION AND WILL HAVE TO BE MODIFIED PER +++++++++++++*)

(*+++++++++++VALVE BANK 1 +++++++++++++*)
(*+++++++++++VALVE BANK 1 +++++++++++++*)
(*+++++++++++VALVE BANK 1 +++++++++++++*)


	(*Valve 1, Model 524 ONLY*)
	(*Clamp #6, 20*)
		Valve1FB
			(
			Enable_Motion:= Enable_Motion ,
			Enable_Latch:= TRUE,					(*Enabling Runs Valve as detent type (maintained solenoids*)
			Enable_SideA_PreCharge:= FALSE,		(*Enabling Turns Side A PreCharge Active, reset when Side B is energized in Auto*)
			Enable_SideB_PreCharge:= FALSE,		(*Enabling Turns Side B PreCharge Active, reset when Side A is energized in Auto*)
			PreCharge_Time:= T#0.1S,
			Enable_Auto_Commands:= In_Auto,
			Enable_Manual_Commands:= In_Manual AND (All_Robots_Clear OR TurntableA_At_Robot),  (*TLK ADDED OR*)
			In_Manual_SideA_Command:= Discrete_In.ManReqs.0,
			In_Manual_SideB_Command:= (Discrete_In.ManReqs.1 OR Discrete_In.Go_Home),
			SideA_Indicator:= (Clamp6ADVD AND Clamp20ADVD),
			SideB_Indicator:= (Clamp6RETD AND Clamp20RETD) OR Manual_Ind_HomePrompt,
			TurnOn_SideA_SOL=> N100.Q.0,
			TurnOn_SideB_SOL=> N100.Q.1,
			TurnOn_SideA_Indicator=> Manual_Indicators1.0,
			TurnOn_SideB_Indicator=> Manual_Indicators1.1
			 );
	IF (Model_ID=2) THEN		 
			Valve1FB.In_Auto_SideA_Command:= Clamp_Step.1 AND NOT Unclamp_Step.0;
			Valve1FB.In_Auto_SideB_Command:= Unclamp_Step.0 
										OR ((TurntableA_At_Robot OR Turntable_Bypassed) AND All_Sensors_Off AND Weld_Robots_Clear);
		ELSE
			Valve1FB.In_Auto_SideA_Command:= FALSE;
			Valve1FB.In_Auto_SideB_Command:= TRUE;
		END_IF

	(*Valve 2, Model 524 ONLY*)
	(*Pin #5, 15*)
		Valve2FB
			(
			Enable_Motion:= Enable_Motion ,
			Enable_Latch:= TRUE,					(*Enabling Runs Valve as detent type (maintained solenoids*)
			Enable_SideA_PreCharge:= FALSE,		(*Enabling Turns Side A PreCharge Active, reset when Side B is energized in Auto*)
			Enable_SideB_PreCharge:= FALSE,		(*Enabling Turns Side B PreCharge Active, reset when Side A is energized in Auto*)
			PreCharge_Time:= T#0.10S,
			Enable_Auto_Commands:= In_Auto,
			Enable_Manual_Commands:= In_Manual AND (All_Robots_Clear OR TurntableA_At_Robot),  (*TLK ADDED OR*)
			In_Manual_SideA_Command:=  Discrete_In.ManReqs.2 ,
			In_Manual_SideB_Command:= (Discrete_In.ManReqs.3 OR Discrete_In.Go_Home),
			SideA_Indicator:=  Pin5ADVD AND Pin15ADVD,
			SideB_Indicator:= (Pin5RETD AND Pin15RETD) OR Manual_Ind_HomePrompt,
			TurnOn_SideA_SOL=> N100.Q.2,
			TurnOn_SideB_SOL=> N100.Q.3,
			TurnOn_SideA_Indicator=> Manual_Indicators1.2,
			TurnOn_SideB_Indicator=> Manual_Indicators1.3
			 );
	IF (Model_ID=2) THEN		 
			Valve2FB.In_Auto_SideA_Command:= Clamp_Step.0 AND NOT Unclamp_Step.1
										OR ((TurntableA_At_Robot OR Turntable_Bypassed) AND All_Sensors_Off AND Weld_Robots_Clear);
			Valve2FB.In_Auto_SideB_Command:= Unclamp_Step.1;
		ELSE
			Valve2FB.In_Auto_SideA_Command:= FALSE;
			Valve2FB.In_Auto_SideB_Command:= TRUE;
		END_IF

	(*Valve 3, Model 524 ONLY*)
	(*Slide #4, 11*)
		Valve3FB
			(
			Enable_Motion:= Enable_Motion ,
			Enable_Latch:= TRUE,					(*Enabling Runs Valve as detent type (maintained solenoids*)
			Enable_SideA_PreCharge:= FALSE,		(*Enabling Turns Side A PreCharge Active, reset when Side B is energized in Auto*)
			Enable_SideB_PreCharge:= FALSE,		(*Enabling Turns Side B PreCharge Active, reset when Side A is energized in Auto*)
			PreCharge_Time:= T#0.10S,
			Enable_Auto_Commands:= In_Auto,
			Enable_Manual_Commands:= In_Manual AND (All_Robots_Clear OR TurntableA_At_Robot),  (*TLK ADDED OR*)
			In_Manual_SideA_Command:= Discrete_In.ManReqs.4,
			In_Manual_SideB_Command:= (Discrete_In.ManReqs.5 OR Discrete_In.Go_Home),
			SideA_Indicator:= Slide4ADVD AND Slide11ADVD,
			SideB_Indicator:= (Slide4RETD AND Slide11RETD) OR Manual_Ind_HomePrompt,
			TurnOn_SideA_SOL=> N100.Q.4,
			TurnOn_SideB_SOL=> N100.Q.5,
			TurnOn_SideA_Indicator=> Manual_Indicators1.4,
			TurnOn_SideB_Indicator=> Manual_Indicators1.5
			 );
	IF (Model_ID=2) THEN
			Valve3FB.In_Auto_SideA_Command:= Clamp_Step.3 AND NOT Unclamp_Step.2;
			Valve3FB.In_Auto_SideB_Command:= Unclamp_Step.2
										OR ((TurntableA_At_Robot OR Turntable_Bypassed) AND All_Sensors_Off AND Weld_Robots_Clear);
		ELSE
			Valve3FB.In_Auto_SideA_Command:= FALSE;
			Valve3FB.In_Auto_SideB_Command:= TRUE;
		END_IF

	(*Valve 4, Model 543 ONLY*)
	(*Clamp #8, 19*)
		Valve4FB
			(
			Enable_Motion:= Enable_Motion ,
			Enable_Latch:= TRUE,					(*Enabling Runs Valve as detent type (maintained solenoids*)
			Enable_SideA_PreCharge:= FALSE,		(*Enabling Turns Side A PreCharge Active, reset when Side B is energized in Auto*)
			Enable_SideB_PreCharge:= FALSE,		(*Enabling Turns Side B PreCharge Active, reset when Side A is energized in Auto*)
			PreCharge_Time:= T#0.10S,
			Enable_Auto_Commands:= In_Auto,
			Enable_Manual_Commands:= In_Manual AND (All_Robots_Clear OR TurntableA_At_Robot),  (*TLK ADDED OR*)
			In_Manual_SideA_Command:= Discrete_In.ManReqs.6,
			In_Manual_SideB_Command:= (Discrete_In.ManReqs.7 OR Discrete_In.Go_Home),
			SideA_Indicator:= Clamp8ADVD AND Clamp19ADVD,
			SideB_Indicator:= (Clamp8RETD AND Clamp19RETD) OR Manual_Ind_HomePrompt,
			TurnOn_SideA_SOL=> N100.Q.6,
			TurnOn_SideB_SOL=> N100.Q.7,
			TurnOn_SideA_Indicator=> Manual_Indicators1.6,
			TurnOn_SideB_Indicator=> Manual_Indicators1.7
			 );
	IF (Model_ID=3) THEN
			Valve4FB.In_Auto_SideA_Command:= Clamp_Step.1 AND NOT Unclamp_Step.0;
			Valve4FB.In_Auto_SideB_Command:= Unclamp_Step.0
										OR ((TurntableA_At_Robot OR Turntable_Bypassed) AND All_Sensors_Off AND Weld_Robots_Clear);
		ELSE
			Valve4FB.In_Auto_SideA_Command:= FALSE;
			Valve4FB.In_Auto_SideB_Command:= TRUE;
		END_IF

	(*Valve 5, Model 543 ONLY*)
	(*Pin #6, 14*)
		Valve5FB
			(
			Enable_Motion:= Enable_Motion ,
			Enable_Latch:= TRUE,					(*Enabling Runs Valve as detent type (maintained solenoids*)
			Enable_SideA_PreCharge:= FALSE,		(*Enabling Turns Side A PreCharge Active, reset when Side B is energized in Auto*)
			Enable_SideB_PreCharge:= FALSE,		(*Enabling Turns Side B PreCharge Active, reset when Side A is energized in Auto*)
			PreCharge_Time:= T#0.10S,
			Enable_Auto_Commands:= In_Auto,
			Enable_Manual_Commands:= In_Manual AND (All_Robots_Clear OR TurntableA_At_Robot),  (*TLK ADDED OR*)
			In_Manual_SideA_Command:= Discrete_In.ManReqs.8,
			In_Manual_SideB_Command:= (Discrete_In.ManReqs.9 OR Discrete_In.Go_Home),
			SideA_Indicator:=  Pin6ADVD AND Pin14ADVD,
			SideB_Indicator:= (Pin6RETD AND Pin14RETD) OR Manual_Ind_HomePrompt,
			TurnOn_SideA_SOL=> N100.Q.8,
			TurnOn_SideB_SOL=> N100.Q.9,
			TurnOn_SideA_Indicator=> Manual_Indicators1.8,
			TurnOn_SideB_Indicator=> Manual_Indicators1.9
			 );
	IF (Model_ID=3) THEN		 
			Valve5FB.In_Auto_SideA_Command:= Clamp_Step.0 AND NOT Unclamp_Step.1
										OR ((TurntableA_At_Robot OR Turntable_Bypassed) AND All_Sensors_Off AND Weld_Robots_Clear);
			Valve5FB.In_Auto_SideB_Command:= Unclamp_Step.1;
		ELSE
			Valve5FB.In_Auto_SideA_Command:= FALSE;
			Valve5FB.In_Auto_SideB_Command:= TRUE;
		END_IF

	(*Valve 6, Model 543 ONLY*)
	(*Swing #1, 3*)
		Valve6FB
			(
			Enable_Motion:= Enable_Motion ,
			Enable_Latch:= TRUE,					(*Enabling Runs Valve as detent type (maintained solenoids*)
			Enable_SideA_PreCharge:= FALSE,		(*Enabling Turns Side A PreCharge Active, reset when Side B is energized in Auto*)
			Enable_SideB_PreCharge:= FALSE,		(*Enabling Turns Side B PreCharge Active, reset when Side A is energized in Auto*)
			PreCharge_Time:= T#0.10S,
			Enable_Auto_Commands:= In_Auto,
			Enable_Manual_Commands:= In_Manual AND (All_Robots_Clear OR TurntableA_At_Robot),  (*TLK ADDED OR*)
			In_Manual_SideA_Command:= Discrete_In.ManReqs.10,
			In_Manual_SideB_Command:= (Discrete_In.ManReqs.11 OR Discrete_In.Go_Home),
			SideA_Indicator:= Swing1ADVD AND Swing3ADVD,
			SideB_Indicator:= (Swing1RETD AND Swing3RETD) OR Manual_Ind_HomePrompt,
			TurnOn_SideA_SOL=> N100.Q.10,
			TurnOn_SideB_SOL=> N100.Q.11,
			TurnOn_SideA_Indicator=> Manual_Indicators1.10,
			TurnOn_SideB_Indicator=> Manual_Indicators1.11
			 );
	IF (Model_ID=3) THEN
			Valve6FB.In_Auto_SideA_Command:= Clamp_Step.3 AND NOT Unclamp_Step.2;
			Valve6FB.In_Auto_SideB_Command:= Unclamp_Step.2
										OR ((TurntableA_At_Robot OR Turntable_Bypassed) AND All_Sensors_Off AND Weld_Robots_Clear);
		ELSE
			Valve6FB.In_Auto_SideA_Command:= FALSE;
			Valve6FB.In_Auto_SideB_Command:= TRUE;
		END_IF

	(*Valve 7, Common*)
	(*Clamp #3, 18 - Manual Clamps*)
		Valve7FB
			(
			Enable_Motion:= Enable_Motion ,
			Enable_Latch:= (TurnTable_WorkingOK OR TurnTableB_At_Robot),					(*Enabling Runs Valve as detent type (maintained solenoids*)
			Enable_SideA_PreCharge:= FALSE,		(*Enabling Turns Side A PreCharge Active, reset when Side B is energized in Auto*)
			Enable_SideB_PreCharge:= FALSE,		(*Enabling Turns Side B PreCharge Active, reset when Side A is energized in Auto*)
			PreCharge_Time:= T#0.10S,
			Enable_Auto_Commands:= In_Auto,
			Enable_Manual_Commands:= In_Manual AND (All_Robots_Clear OR TurntableA_At_Robot),  (*TLK ADDED OR*)
			In_Manual_SideA_Command:= Discrete_In.ManReqs.12,
			In_Manual_SideB_Command:= (Discrete_In.ManReqs.13 OR Discrete_In.Go_Home),
			SideA_Indicator:= Clamp3ADVD AND Clamp18ADVD,
			SideB_Indicator:= (Clamp3RETD AND Clamp18RETD) OR Manual_Ind_HomePrompt,
			TurnOn_SideA_SOL=> N100.Q.12,
			TurnOn_SideB_SOL=> N100.Q.13,
			TurnOn_SideA_Indicator=> Manual_Indicators1.12,
			TurnOn_SideB_Indicator=> Manual_Indicators1.13
			 );
		Valve7FB.In_Auto_SideA_Command:= Clamp_Step.1 AND NOT Unclamp_Step.0;
		Valve7FB.In_Auto_SideB_Command:= Unclamp_Step.0
										OR ((TurntableA_At_Robot OR Turntable_Bypassed) AND All_Sensors_Off AND Weld_Robots_Clear);


	(*Valve 8, Common*)
	(*Pin #1-4, 7, 9, 16-18, Slide #10*)
		Valve8FB
			(
			Enable_Motion:= Enable_Motion ,
			Enable_Latch:= TRUE,					(*Enabling Runs Valve as detent type (maintained solenoids*)
			Enable_SideA_PreCharge:= FALSE,		(*Enabling Turns Side A PreCharge Active, reset when Side B is energized in Auto*)
			Enable_SideB_PreCharge:= FALSE,		(*Enabling Turns Side B PreCharge Active, reset when Side A is energized in Auto*)
			PreCharge_Time:= T#0.10S,
			Enable_Auto_Commands:= In_Auto,
			Enable_Manual_Commands:= In_Manual AND (All_Robots_Clear OR TurntableA_At_Robot),  (*TLK ADDED OR*)
			In_Manual_SideA_Command:= (Discrete_In.ManReqs.14 OR Discrete_In.Go_Home),
			In_Manual_SideB_Command:= Discrete_In.ManReqs.15,
			SideA_Indicator:= (Pin1ADVD AND Pin2ADVD AND Pin3ADVD AND Pin4ADVD AND Pin7ADVD AND Pin9ADVD AND Pin16ADVD AND Pin17ADVD AND Pin18ADVD AND Slide10ADVD) OR Manual_Ind_HomePrompt,
			SideB_Indicator:= Pin1RETD AND Pin2RETD AND Pin3RETD AND Pin4RETD AND Pin7RETD AND Pin9RETD AND Pin16RETD AND Pin17RETD AND Pin18RETD AND Slide10RETD,
			TurnOn_SideA_SOL=> N100.Q.14,
			TurnOn_SideB_SOL=> N100.Q.15,
			TurnOn_SideA_Indicator=> Manual_Indicators1.14,
			TurnOn_SideB_Indicator=> Manual_Indicators1.15
			 );
		Valve8FB.In_Auto_SideA_Command:= Clamp_Step.0 AND NOT Unclamp_Step.1
										OR ((TurntableA_At_Robot OR Turntable_Bypassed) AND All_Sensors_Off AND Weld_Robots_Clear);
		Valve8FB.In_Auto_SideB_Command:= Unclamp_Step.1;


	(*Valve 9, Common*)
	(*Clamp #1, 2, 4, 5, 10, 14, 21, 22*)
		Valve9FB
			(
			Enable_Motion:= Enable_Motion ,
			Enable_Latch:= TRUE,					(*Enabling Runs Valve as detent type (maintained solenoids*)
			Enable_SideA_PreCharge:= FALSE,		(*Enabling Turns Side A PreCharge Active, reset when Side B is energized in Auto*)
			Enable_SideB_PreCharge:= FALSE,		(*Enabling Turns Side B PreCharge Active, reset when Side A is energized in Auto*)
			PreCharge_Time:= T#0.10S,
			Enable_Auto_Commands:= In_Auto,
			Enable_Manual_Commands:= In_Manual AND (All_Robots_Clear OR TurntableA_At_Robot),  (*TLK ADDED OR*)
			In_Manual_SideA_Command:= Discrete_In.ManReqs.16,
			In_Manual_SideB_Command:= (Discrete_In.ManReqs.17 OR Discrete_In.Go_Home),
			SideA_Indicator:= Clamp1ADVD AND Clamp2ADVD AND Clamp4ADVD AND Clamp5ADVD AND Clamp10ADVD AND Clamp14ADVD AND Clamp21ADVD AND Clamp22ADVD,
			SideB_Indicator:= (Clamp1RETD AND Clamp2RETD AND Clamp4RETD AND Clamp5RETD AND Clamp10RETD AND Clamp14RETD AND Clamp21RETD AND Clamp22RETD) OR Manual_Ind_HomePrompt,
			TurnOn_SideA_SOL=> N100.Q.16,
			TurnOn_SideB_SOL=> N100.Q.17,
			TurnOn_SideA_Indicator=> Manual_Indicators1.16,
			TurnOn_SideB_Indicator=> Manual_Indicators1.17
			 );
		Valve9FB.In_Auto_SideA_Command:= Clamp_Step.1 AND NOT Unclamp_Step.0;
		Valve9FB.In_Auto_SideB_Command:= Unclamp_Step.0
										OR ((TurntableA_At_Robot OR Turntable_Bypassed) AND All_Sensors_Off AND Weld_Robots_Clear);


	(*Valve 10, Common*)
	(*Pin #8, 10-13, Slide #1, 2, 13, 14*)
		Valve10FB
			(
			Enable_Motion:= Enable_Motion ,
			Enable_Latch:= TRUE,					(*Enabling Runs Valve as detent type (maintained solenoids*)
			Enable_SideA_PreCharge:= FALSE,		(*Enabling Turns Side A PreCharge Active, reset when Side B is energized in Auto*)
			Enable_SideB_PreCharge:= FALSE,		(*Enabling Turns Side B PreCharge Active, reset when Side A is energized in Auto*)
			PreCharge_Time:= T#0.10S,
			Enable_Auto_Commands:= In_Auto,
			Enable_Manual_Commands:= In_Manual AND (All_Robots_Clear OR TurntableA_At_Robot),  (*TLK ADDED OR*)
			In_Manual_SideA_Command:= (Discrete_In.ManReqs.18 OR Discrete_In.Go_Home),
			In_Manual_SideB_Command:= Discrete_In.ManReqs.19,
			SideA_Indicator:= (Pin8ADVD AND Pin10ADVD AND Pin11ADVD AND Pin12ADVD AND Pin13ADVD AND Slide1ADVD AND Slide2ADVD AND Slide13ADVD AND Slide14ADVD) OR Manual_Ind_HomePrompt,
			SideB_Indicator:= Pin8RETD AND Pin10RETD AND Pin11RETD AND Pin12RETD AND Pin13RETD AND Slide1RETD AND Slide2RETD AND Slide13RETD AND Slide14RETD,
			TurnOn_SideA_SOL=> N100.Q.18,
			TurnOn_SideB_SOL=> N100.Q.19,
			TurnOn_SideA_Indicator=> Manual_Indicators1.18,
			TurnOn_SideB_Indicator=> Manual_Indicators1.19
			 );
		Valve10FB.In_Auto_SideA_Command:= Clamp_Step.0 AND NOT Unclamp_Step.1
										OR ((TurntableA_At_Robot OR Turntable_Bypassed) AND All_Sensors_Off AND Weld_Robots_Clear);
		Valve10FB.In_Auto_SideB_Command:= Unclamp_Step.1;


	(*Valve 11, Common*)
	(*Clamp #9, 12, 13, 16*)
		Valve11FB
			(
			Enable_Motion:= Enable_Motion ,
			Enable_Latch:= TRUE,					(*Enabling Runs Valve as detent type (maintained solenoids*)
			Enable_SideA_PreCharge:= FALSE,		(*Enabling Turns Side A PreCharge Active, reset when Side B is energized in Auto*)
			Enable_SideB_PreCharge:= FALSE,		(*Enabling Turns Side B PreCharge Active, reset when Side A is energized in Auto*)
			PreCharge_Time:= T#0.10S,
			Enable_Auto_Commands:= In_Auto,
			Enable_Manual_Commands:= In_Manual AND (All_Robots_Clear OR TurntableA_At_Robot),  (*TLK ADDED OR*)
			In_Manual_SideA_Command:= Discrete_In.ManReqs.20,
			In_Manual_SideB_Command:= (Discrete_In.ManReqs.21 OR Discrete_In.Go_Home),
			SideA_Indicator:= Clamp9ADVD AND Clamp12ADVD AND Clamp13ADVD AND Clamp16ADVD,
			SideB_Indicator:= (Clamp9RETD AND Clamp12RETD AND Clamp13RETD AND Clamp16RETD) OR Manual_Ind_HomePrompt,
			TurnOn_SideA_SOL=> N100.Q.20,
			TurnOn_SideB_SOL=> N100.Q.21,
			TurnOn_SideA_Indicator=> Manual_Indicators1.20,
			TurnOn_SideB_Indicator=> Manual_Indicators1.21
			 );
		Valve11FB.In_Auto_SideA_Command:= Clamp_Step.1 AND NOT Unclamp_Step.0;
		Valve11FB.In_Auto_SideB_Command:= Unclamp_Step.0
										OR ((TurntableA_At_Robot OR Turntable_Bypassed) AND All_Sensors_Off AND Weld_Robots_Clear);


	(*Valve 12, Common*)
	(*Slide #3, 5, 7-9, 12, Swing #2*)
		Valve12FB
			(
			Enable_Motion:= Enable_Motion,
			Enable_Latch:= TRUE,					(*Enabling Runs Valve as detent type (maintained solenoids*)
			Enable_SideA_PreCharge:= FALSE,		(*Enabling Turns Side A PreCharge Active, reset when Side B is energized in Auto*)
			Enable_SideB_PreCharge:= FALSE,		(*Enabling Turns Side B PreCharge Active, reset when Side A is energized in Auto*)
			PreCharge_Time:= T#0.10S,
			Enable_Auto_Commands:= In_Auto,
			Enable_Manual_Commands:= In_Manual AND (All_Robots_Clear OR TurntableA_At_Robot),  (*TLK ADDED OR*)
			In_Manual_SideA_Command:= Discrete_In.ManReqs.22,
			In_Manual_SideB_Command:= (Discrete_In.ManReqs.23 OR Discrete_In.Go_Home),
			SideA_Indicator:= Slide3ADVD AND Slide5ADVD AND Slide7ADVD AND Slide8ADVD AND Slide9ADVD AND Slide12ADVD AND Swing2ADVD,
			SideB_Indicator:= (Slide3RETD AND Slide5RETD AND Slide7RETD AND Slide8RETD AND Slide9RETD AND Slide12RETD AND Swing2RETD) OR Manual_Ind_HomePrompt,
			TurnOn_SideA_SOL=> N100.Q.22,
			TurnOn_SideB_SOL=> N100.Q.23,
			TurnOn_SideA_Indicator=> Manual_Indicators1.22,
			TurnOn_SideB_Indicator=> Manual_Indicators1.23
			 );
		Valve12FB.In_Auto_SideA_Command:= Clamp_Step.3 AND NOT Unclamp_Step.2;
		Valve12FB.In_Auto_SideB_Command:= Unclamp_Step.2
										OR ((TurntableA_At_Robot OR Turntable_Bypassed) AND All_Sensors_Off AND Weld_Robots_Clear);


	(*Valve 13, Common*)
	(*Clamp #7, 11, 15, 17*)
		Valve13FB
			(
			Enable_Motion:= Enable_Motion,
			Enable_Latch:= TRUE,					(*Enabling Runs Valve as detent type (maintained solenoids*)
			Enable_SideA_PreCharge:= FALSE,		(*Enabling Turns Side A PreCharge Active, reset when Side B is energized in Auto*)
			Enable_SideB_PreCharge:= FALSE,		(*Enabling Turns Side B PreCharge Active, reset when Side A is energized in Auto*)
			PreCharge_Time:= T#0.10S,
			Enable_Auto_Commands:= In_Auto,
			Enable_Manual_Commands:= In_Manual AND (All_Robots_Clear OR TurntableA_At_Robot),  (*TLK ADDED OR*)
			In_Manual_SideA_Command:= Discrete_In.ManReqs.24,
			In_Manual_SideB_Command:= (Discrete_In.ManReqs.25 OR Discrete_In.Go_Home),
			SideA_Indicator:= Clamp7ADVD AND Clamp11ADVD AND Clamp15ADVD AND Clamp17ADVD,
			SideB_Indicator:= (Clamp7RETD AND Clamp11RETD AND Clamp15RETD AND Clamp17RETD) OR Manual_Ind_HomePrompt,
			TurnOn_SideA_SOL=> N100.Q.24,
			TurnOn_SideB_SOL=> N100.Q.25,
			TurnOn_SideA_Indicator=> Manual_Indicators1.24,
			TurnOn_SideB_Indicator=> Manual_Indicators1.25
			 );
		Valve13FB.In_Auto_SideA_Command:= Clamp_Step.2 AND NOT Unclamp_Step.3;
		Valve13FB.In_Auto_SideB_Command:= Unclamp_Step.3
										OR ((TurntableA_At_Robot OR Turntable_Bypassed) AND All_Sensors_Off AND Weld_Robots_Clear);	
		
		
	(*Valve 14, A+B*)
	(*Locks*)
		Valve14FB
			(
			Enable_Motion:= Enable_Motion ,
			Enable_Latch:= FALSE,					(*Enabling Runs Valve as detent type (maintained solenoids*)
			Enable_SideA_PreCharge:= FALSE,		(*Enabling Turns Side A PreCharge Active, reset when Side B is energized in Auto*)
			Enable_SideB_PreCharge:= FALSE,		(*Enabling Turns Side B PreCharge Active, reset when Side A is energized in Auto*)
			PreCharge_Time:= T#0.10S,
			Enable_Auto_Commands:= In_Auto,
			Enable_Manual_Commands:= In_Manual AND (All_Robots_Clear OR TurntableA_At_Robot),
			In_Manual_SideA_Command:= Discrete_In.ManReqs.26,
			In_Manual_SideB_Command:= Discrete_In.ManReqs.27 
										OR (N100.Q.5 AND NOT (Slide4RETD AND Slide11RETD)) 
										OR (N100.Q.15 AND NOT Slide10RETD) 
										OR (N100.Q.19 AND NOT (Slide1RETD AND Slide2RETD AND Slide13RETD AND Slide14RETD))
										OR (N100.Q.23 AND NOT (Slide3RETD AND Slide5RETD AND Slide7RETD AND Slide8RETD AND Slide9RETD AND Slide12RETD))
										OR (N100.Q.28 AND NOT Slide6RETD)
										OR (N100.Q.4 AND NOT (Slide4ADVD AND Slide11ADVD)) 
										OR (N100.Q.14 AND NOT Slide10ADVD) 
										OR (N100.Q.18 AND NOT (Slide1ADVD AND Slide2ADVD AND Slide13ADVD AND Slide14ADVD))
										OR (N100.Q.22 AND NOT (Slide3ADVD AND Slide5ADVD AND Slide7ADVD AND Slide8ADVD AND Slide9ADVD AND Slide12ADVD))
										OR (N100.Q.28 AND NOT Slide6ADVD),
			SideA_Indicator:= FALSE,
			SideB_Indicator:= FALSE,
			TurnOn_SideA_SOL=> N100.Q.26,
			TurnOn_SideB_SOL=> N100.Q.27,
			TurnOn_SideA_Indicator=> Manual_Indicators1.26,
			TurnOn_SideB_Indicator=> Manual_Indicators1.27
			 );
		Valve14FB.In_Auto_SideA_Command:= NOT Valve14FB.In_Auto_SideB_Command;
		Valve14FB.In_Auto_SideB_Command:= (N100.Q.5 AND NOT (Slide4RETD AND Slide11RETD)) 
										OR (N100.Q.15 AND NOT Slide10RETD) 
										OR (N100.Q.19 AND NOT (Slide1RETD AND Slide2RETD AND Slide13RETD AND Slide14RETD))
										OR (N100.Q.23 AND NOT (Slide3RETD AND Slide5RETD AND Slide7RETD AND Slide8RETD AND Slide9RETD AND Slide12RETD))
										OR (N100.Q.29 AND NOT Slide6RETD)
										OR (N100.Q.4 AND NOT (Slide4ADVD AND Slide11ADVD)) 
										OR (N100.Q.14 AND NOT Slide10ADVD) 
										OR (N100.Q.18 AND NOT (Slide1ADVD AND Slide2ADVD AND Slide13ADVD AND Slide14ADVD))
										OR (N100.Q.22 AND NOT (Slide3ADVD AND Slide5ADVD AND Slide7ADVD AND Slide8ADVD AND Slide9ADVD AND Slide12ADVD))
										OR (N100.Q.28 AND NOT Slide6ADVD);

	(*Valve 15, A+B*)
	(*Slide #6*)
		Valve15FB
			(
			Enable_Motion:= Enable_Motion ,
			Enable_Latch:= TRUE,					(*Enabling Runs Valve as detent type (maintained solenoids*)
			Enable_SideA_PreCharge:= FALSE,		(*Enabling Turns Side A PreCharge Active, reset when Side B is energized in Auto*)
			Enable_SideB_PreCharge:= FALSE,		(*Enabling Turns Side B PreCharge Active, reset when Side A is energized in Auto*)
			PreCharge_Time:= T#0.10S,
			Enable_Auto_Commands:= In_Auto,
			Enable_Manual_Commands:= In_Manual AND (All_Robots_Clear OR TurntableA_At_Robot),  (*TLK ADDED OR*)
			In_Manual_SideA_Command:= Discrete_In.ManReqs.28,
			In_Manual_SideB_Command:= Discrete_In.ManReqs.29,
			SideA_Indicator:= Slide6ADVD,
			SideB_Indicator:= Slide6RETD,
			TurnOn_SideA_SOL=> N100.Q.28,
			TurnOn_SideB_SOL=> N100.Q.29,
			TurnOn_SideA_Indicator=> Manual_Indicators1.28,
			TurnOn_SideB_Indicator=> Manual_Indicators1.29
			 );
		Valve15FB.In_Auto_SideA_Command:= Clamp_Step.3 AND NOT Unclamp_Step.2;
		Valve15FB.In_Auto_SideB_Command:= ((TurntableA_At_Robot OR Turntable_Bypassed) AND All_Sensors_Off AND Weld_Robots_Clear);
		
		
(*--------------------------------------------------------------------------------------------------------------------------------------------*)		
(*                                                           Spare Valves                                                                     *)
(*--------------------------------------------------------------------------------------------------------------------------------------------*)


	(*Valve 16, A+B*)
	(*spare*)
		Valve16FB
			(
			Enable_Motion:= Enable_Motion ,
			Enable_Latch:= TRUE,					(*Enabling Runs Valve as detent type (maintained solenoids*)
			Enable_SideA_PreCharge:= FALSE,		(*Enabling Turns Side A PreCharge Active, reset when Side B is energized in Auto*)
			Enable_SideB_PreCharge:= FALSE,		(*Enabling Turns Side B PreCharge Active, reset when Side A is energized in Auto*)
			PreCharge_Time:= T#0.10S,
			Enable_Auto_Commands:= In_Auto,
			Enable_Manual_Commands:= In_Manual AND (All_Robots_Clear OR TurntableA_At_Robot),  (*TLK ADDED OR*)
			In_Manual_SideA_Command:= Discrete_In.ManReqs.30,
			In_Manual_SideB_Command:= Discrete_In.ManReqs.31,
			SideA_Indicator:= FALSE,
			SideB_Indicator:= FALSE,
			TurnOn_SideA_SOL=> N100.Q.30,
			TurnOn_SideB_SOL=> N100.Q.31,
			TurnOn_SideA_Indicator=> Manual_Indicators1.30,
			TurnOn_SideB_Indicator=> Manual_Indicators1.31
			 );
		Valve16FB.In_Auto_SideA_Command:= FALSE;
		Valve16FB.In_Auto_SideB_Command:= FALSE;


























(*end*)
END_ACTION

ACTION ValveBank2:


(*+++++++++++THIS AREA IS CUSTOM PER INSTALLATION AND WILL HAVE TO BE MODIFIED PER +++++++++++++*)
(*+++++++++++THIS AREA IS CUSTOM PER INSTALLATION AND WILL HAVE TO BE MODIFIED PER +++++++++++++*)
(*+++++++++++THIS AREA IS CUSTOM PER INSTALLATION AND WILL HAVE TO BE MODIFIED PER +++++++++++++*)

(*+++++++++++VALVE BANK 2 +++++++++++++*)
(*+++++++++++VALVE BANK 2 +++++++++++++*)
(*+++++++++++VALVE BANK 2 +++++++++++++*)


	(*Valve 17, A+B*)
	(*spare*)
		Valve17FB
			(
			Enable_Motion:= Enable_Motion ,
			Enable_Latch:= TRUE,					(*Enabling Runs Valve as detent type (maintained solenoids*)
			Enable_SideA_PreCharge:= FALSE,		(*Enabling Turns Side A PreCharge Active, reset when Side B is energized in Auto*)
			Enable_SideB_PreCharge:= FALSE,		(*Enabling Turns Side B PreCharge Active, reset when Side A is energized in Auto*)
			PreCharge_Time:= T#0.1S,
			Enable_Auto_Commands:= In_Auto,
			Enable_Manual_Commands:= In_Manual AND All_Robots_Clear,
			In_Manual_SideA_Command:= Discrete_In.ManReqs2.0,
			In_Manual_SideB_Command:= (Discrete_In.ManReqs2.1 OR Discrete_In.Go_Home),
			SideA_Indicator:= FALSE,
			SideB_Indicator:= FALSE,
			TurnOn_SideA_SOL=> N101.Q.0,
			TurnOn_SideB_SOL=> N101.Q.1,
			TurnOn_SideA_Indicator=> Manual_Indicators2.0,
			TurnOn_SideB_Indicator=> Manual_Indicators2.1
			 );
		Valve17FB.In_Auto_SideA_Command:= FALSE;
		Valve17FB.In_Auto_SideB_Command:= FALSE;


	(*Valve 18, A+B*)
	(*spare*)
		Valve18FB
			(
			Enable_Motion:= Enable_Motion ,
			Enable_Latch:= TRUE,					(*Enabling Runs Valve as detent type (maintained solenoids*)
			Enable_SideA_PreCharge:= FALSE,		(*Enabling Turns Side A PreCharge Active, reset when Side B is energized in Auto*)
			Enable_SideB_PreCharge:= FALSE,		(*Enabling Turns Side B PreCharge Active, reset when Side A is energized in Auto*)
			PreCharge_Time:= T#0.10S,
			Enable_Auto_Commands:= In_Auto,
			Enable_Manual_Commands:= In_Manual AND All_Robots_Clear,
			In_Manual_SideA_Command:= Discrete_In.ManReqs2.2,
			In_Manual_SideB_Command:= Discrete_In.ManReqs2.3,
			SideA_Indicator:= FALSE,
			SideB_Indicator:= FALSE,
			TurnOn_SideA_SOL=> N101.Q.2,
			TurnOn_SideB_SOL=> N101.Q.3,
			TurnOn_SideA_Indicator=> Manual_Indicators2.2,
			TurnOn_SideB_Indicator=> Manual_Indicators2.3
			 );
		Valve18FB.In_Auto_SideA_Command:= FALSE;
		Valve18FB.In_Auto_SideB_Command:= FALSE;

	(*Valve 19, A+B*)
	(*spare*)
		Valve19FB
			(
			Enable_Motion:= Enable_Motion ,
			Enable_Latch:= TRUE,					(*Enabling Runs Valve as detent type (maintained solenoids*)
			Enable_SideA_PreCharge:= FALSE,		(*Enabling Turns Side A PreCharge Active, reset when Side B is energized in Auto*)
			Enable_SideB_PreCharge:= FALSE,		(*Enabling Turns Side B PreCharge Active, reset when Side A is energized in Auto*)
			PreCharge_Time:= T#0.10S,
			Enable_Auto_Commands:= In_Auto,
			Enable_Manual_Commands:= In_Manual AND All_Robots_Clear,
			In_Manual_SideA_Command:= Discrete_In.ManReqs2.4,
			In_Manual_SideB_Command:= Discrete_In.ManReqs2.5,
			SideA_Indicator:= FALSE,
			SideB_Indicator:= FALSE,
			TurnOn_SideA_SOL=> N101.Q.4,
			TurnOn_SideB_SOL=> N101.Q.5,
			TurnOn_SideA_Indicator=> Manual_Indicators2.4,
			TurnOn_SideB_Indicator=> Manual_Indicators2.5
			 );
		Valve19FB.In_Auto_SideA_Command:= FALSE;
		Valve19FB.In_Auto_SideB_Command:= FALSE;


	(*Valve 20, A+B*)
	(*spare*)
		Valve20FB
			(
			Enable_Motion:= Enable_Motion ,
			Enable_Latch:= TRUE,					(*Enabling Runs Valve as detent type (maintained solenoids*)
			Enable_SideA_PreCharge:= FALSE,		(*Enabling Turns Side A PreCharge Active, reset when Side B is energized in Auto*)
			Enable_SideB_PreCharge:= FALSE,		(*Enabling Turns Side B PreCharge Active, reset when Side A is energized in Auto*)
			PreCharge_Time:= T#0.10S,
			Enable_Auto_Commands:= In_Auto,
			Enable_Manual_Commands:= In_Manual AND All_Robots_Clear,
			In_Manual_SideA_Command:= Discrete_In.ManReqs2.6,
			In_Manual_SideB_Command:= Discrete_In.ManReqs2.7,
			SideA_Indicator:= FALSE,
			SideB_Indicator:= FALSE,
			TurnOn_SideA_SOL=> N101.Q.6,
			TurnOn_SideB_SOL=> N101.Q.7,
			TurnOn_SideA_Indicator=> Manual_Indicators2.6,
			TurnOn_SideB_Indicator=> Manual_Indicators2.7
			 );
		Valve20FB.In_Auto_SideA_Command:= FALSE;
		Valve20FB.In_Auto_SideB_Command:= FALSE;


	(*Valve 21, A+B*)
	(*spare*)
		Valve21FB
			(
			Enable_Motion:= Enable_Motion ,
			Enable_Latch:= TRUE,					(*Enabling Runs Valve as detent type (maintained solenoids*)
			Enable_SideA_PreCharge:= FALSE,		(*Enabling Turns Side A PreCharge Active, reset when Side B is energized in Auto*)
			Enable_SideB_PreCharge:= FALSE,		(*Enabling Turns Side B PreCharge Active, reset when Side A is energized in Auto*)
			PreCharge_Time:= T#0.10S,
			Enable_Auto_Commands:= In_Auto,
			Enable_Manual_Commands:= In_Manual AND All_Robots_Clear,
			In_Manual_SideA_Command:= Discrete_In.ManReqs2.8,
			In_Manual_SideB_Command:= Discrete_In.ManReqs2.9,
			SideA_Indicator:= FALSE,
			SideB_Indicator:= FALSE,
			TurnOn_SideA_SOL=> N101.Q.8,
			TurnOn_SideB_SOL=> N101.Q.9,
			TurnOn_SideA_Indicator=> Manual_Indicators2.8,
			TurnOn_SideB_Indicator=> Manual_Indicators2.9
			 );
		Valve21FB.In_Auto_SideA_Command:= FALSE;
		Valve21FB.In_Auto_SideB_Command:= FALSE;


	(*Valve 22, A+B*)
	(*spare*)
		Valve22FB
			(
			Enable_Motion:= Enable_Motion ,
			Enable_Latch:= TRUE,					(*Enabling Runs Valve as detent type (maintained solenoids*)
			Enable_SideA_PreCharge:= FALSE,		(*Enabling Turns Side A PreCharge Active, reset when Side B is energized in Auto*)
			Enable_SideB_PreCharge:= FALSE,		(*Enabling Turns Side B PreCharge Active, reset when Side A is energized in Auto*)
			PreCharge_Time:= T#0.10S,
			Enable_Auto_Commands:= In_Auto,
			Enable_Manual_Commands:= In_Manual AND All_Robots_Clear,
			In_Manual_SideA_Command:= Discrete_In.ManReqs2.10,
			In_Manual_SideB_Command:= Discrete_In.ManReqs2.11,
			SideA_Indicator:= FALSE,
			SideB_Indicator:= FALSE,
			TurnOn_SideA_SOL=> N101.Q.10,
			TurnOn_SideB_SOL=> N101.Q.11,
			TurnOn_SideA_Indicator=> Manual_Indicators2.10,
			TurnOn_SideB_Indicator=> Manual_Indicators2.11
			 );
		Valve22FB.In_Auto_SideA_Command:= FALSE;
		Valve22FB.In_Auto_SideB_Command:= FALSE;


	(*Valve 23, A+B*)
	(*spare*)
		Valve23FB
			(
			Enable_Motion:= Enable_Motion ,
			Enable_Latch:= TRUE,					(*Enabling Runs Valve as detent type (maintained solenoids*)
			Enable_SideA_PreCharge:= FALSE,		(*Enabling Turns Side A PreCharge Active, reset when Side B is energized in Auto*)
			Enable_SideB_PreCharge:= FALSE,		(*Enabling Turns Side B PreCharge Active, reset when Side A is energized in Auto*)
			PreCharge_Time:= T#0.10S,
			Enable_Auto_Commands:= In_Auto,
			Enable_Manual_Commands:= In_Manual AND All_Robots_Clear,
			In_Manual_SideA_Command:= Discrete_In.ManReqs2.12,
			In_Manual_SideB_Command:= Discrete_In.ManReqs2.13,
			SideA_Indicator:= FALSE,
			SideB_Indicator:= FALSE,
			TurnOn_SideA_SOL=> N101.Q.12,
			TurnOn_SideB_SOL=> N101.Q.13,
			TurnOn_SideA_Indicator=> Manual_Indicators2.12,
			TurnOn_SideB_Indicator=> Manual_Indicators2.13
			 );
		Valve23FB.In_Auto_SideA_Command:= FALSE;
		Valve23FB.In_Auto_SideB_Command:= FALSE;


	(*Valve 24, A+B*)
	(*spare*)
		Valve24FB
			(
			Enable_Motion:= Enable_Motion ,
			Enable_Latch:= TRUE,					(*Enabling Runs Valve as detent type (maintained solenoids*)
			Enable_SideA_PreCharge:= FALSE,		(*Enabling Turns Side A PreCharge Active, reset when Side B is energized in Auto*)
			Enable_SideB_PreCharge:= FALSE,		(*Enabling Turns Side B PreCharge Active, reset when Side A is energized in Auto*)
			PreCharge_Time:= T#0.10S,
			Enable_Auto_Commands:= In_Auto,
			Enable_Manual_Commands:= In_Manual AND All_Robots_Clear,
			In_Manual_SideA_Command:= Discrete_In.ManReqs2.14,
			In_Manual_SideB_Command:= Discrete_In.ManReqs2.15,
			SideA_Indicator:= FALSE,
			SideB_Indicator:= FALSE,
			TurnOn_SideA_SOL=> N101.Q.14,
			TurnOn_SideB_SOL=> N101.Q.15,
			TurnOn_SideA_Indicator=> Manual_Indicators2.14,
			TurnOn_SideB_Indicator=> Manual_Indicators2.15
			 );
		Valve24FB.In_Auto_SideA_Command:= FALSE;
		Valve24FB.In_Auto_SideB_Command:= FALSE;


	(*Valve 25, A+B*)
	(*spare*)
		Valve25FB
			(
			Enable_Motion:= Enable_Motion ,
			Enable_Latch:= TRUE,					(*Enabling Runs Valve as detent type (maintained solenoids*)
			Enable_SideA_PreCharge:= FALSE,		(*Enabling Turns Side A PreCharge Active, reset when Side B is energized in Auto*)
			Enable_SideB_PreCharge:= FALSE,		(*Enabling Turns Side B PreCharge Active, reset when Side A is energized in Auto*)
			PreCharge_Time:= T#0.10S,
			Enable_Auto_Commands:= In_Auto,
			Enable_Manual_Commands:= In_Manual AND All_Robots_Clear,
			In_Manual_SideA_Command:= Discrete_In.ManReqs2.16,
			In_Manual_SideB_Command:= Discrete_In.ManReqs2.17,
			SideA_Indicator:= FALSE,
			SideB_Indicator:= FALSE,
			TurnOn_SideA_SOL=> N101.Q.16,
			TurnOn_SideB_SOL=> N101.Q.17,
			TurnOn_SideA_Indicator=> Manual_Indicators2.16,
			TurnOn_SideB_Indicator=> Manual_Indicators2.17
			 );
		Valve25FB.In_Auto_SideA_Command:= FALSE;
		Valve25FB.In_Auto_SideB_Command:= FALSE;


	(*Valve 26, A+B*)
	(*spare*)
		Valve26FB
			(
			Enable_Motion:= Enable_Motion ,
			Enable_Latch:= TRUE,					(*Enabling Runs Valve as detent type (maintained solenoids*)
			Enable_SideA_PreCharge:= FALSE,		(*Enabling Turns Side A PreCharge Active, reset when Side B is energized in Auto*)
			Enable_SideB_PreCharge:= FALSE,		(*Enabling Turns Side B PreCharge Active, reset when Side A is energized in Auto*)
			PreCharge_Time:= T#0.10S,
			Enable_Auto_Commands:= In_Auto,
			Enable_Manual_Commands:= In_Manual AND All_Robots_Clear,
			In_Manual_SideA_Command:= Discrete_In.ManReqs2.18,
			In_Manual_SideB_Command:= Discrete_In.ManReqs2.19,
			SideA_Indicator:= FALSE,
			SideB_Indicator:= FALSE,
			TurnOn_SideA_SOL=> N101.Q.18,
			TurnOn_SideB_SOL=> N101.Q.19,
			TurnOn_SideA_Indicator=> Manual_Indicators2.18,
			TurnOn_SideB_Indicator=> Manual_Indicators2.19
			 );
		Valve26FB.In_Auto_SideA_Command:= FALSE;
		Valve26FB.In_Auto_SideB_Command:= FALSE;


	(*Valve 27, A+B*)
	(*spare*)
		Valve27FB
			(
			Enable_Motion:= Enable_Motion ,
			Enable_Latch:= TRUE,					(*Enabling Runs Valve as detent type (maintained solenoids*)
			Enable_SideA_PreCharge:= FALSE,		(*Enabling Turns Side A PreCharge Active, reset when Side B is energized in Auto*)
			Enable_SideB_PreCharge:= FALSE,		(*Enabling Turns Side B PreCharge Active, reset when Side A is energized in Auto*)
			PreCharge_Time:= T#0.10S,
			Enable_Auto_Commands:= In_Auto,
			Enable_Manual_Commands:= In_Manual AND All_Robots_Clear,
			In_Manual_SideA_Command:= Discrete_In.ManReqs2.20,
			In_Manual_SideB_Command:= Discrete_In.ManReqs2.21,
			SideA_Indicator:= FALSE,
			SideB_Indicator:= FALSE,
			TurnOn_SideA_SOL=> N101.Q.20,
			TurnOn_SideB_SOL=> N101.Q.21,
			TurnOn_SideA_Indicator=> Manual_Indicators2.20,
			TurnOn_SideB_Indicator=> Manual_Indicators2.21
			 );
		Valve27FB.In_Auto_SideA_Command:= FALSE;
		Valve27FB.In_Auto_SideB_Command:= FALSE;


	(*Valve 28, A+B*)
	(*spare*)
		Valve28FB
			(
			Enable_Motion:= Enable_Motion ,
			Enable_Latch:= TRUE,					(*Enabling Runs Valve as detent type (maintained solenoids*)
			Enable_SideA_PreCharge:= FALSE,		(*Enabling Turns Side A PreCharge Active, reset when Side B is energized in Auto*)
			Enable_SideB_PreCharge:= FALSE,		(*Enabling Turns Side B PreCharge Active, reset when Side A is energized in Auto*)
			PreCharge_Time:= T#0.10S,
			Enable_Auto_Commands:= In_Auto,
			Enable_Manual_Commands:= In_Manual AND All_Robots_Clear,
			In_Manual_SideA_Command:= Discrete_In.ManReqs2.22,
			In_Manual_SideB_Command:= Discrete_In.ManReqs2.23,
			SideA_Indicator:= FALSE,
			SideB_Indicator:= FALSE,
			TurnOn_SideA_SOL=> N101.Q.22,
			TurnOn_SideB_SOL=> N101.Q.23,
			TurnOn_SideA_Indicator=> Manual_Indicators2.22,
			TurnOn_SideB_Indicator=> Manual_Indicators2.23
			 );
		Valve28FB.In_Auto_SideA_Command:= FALSE;
		Valve28FB.In_Auto_SideB_Command:= FALSE;


	(*Valve 29, A+B*)
	(*spare*)
		Valve29FB
			(
			Enable_Motion:= Enable_Motion ,
			Enable_Latch:= TRUE,					(*Enabling Runs Valve as detent type (maintained solenoids*)
			Enable_SideA_PreCharge:= FALSE,		(*Enabling Turns Side A PreCharge Active, reset when Side B is energized in Auto*)
			Enable_SideB_PreCharge:= FALSE,		(*Enabling Turns Side B PreCharge Active, reset when Side A is energized in Auto*)
			PreCharge_Time:= T#0.10S,
			Enable_Auto_Commands:= In_Auto,
			Enable_Manual_Commands:= In_Manual AND All_Robots_Clear,
			In_Manual_SideA_Command:= Discrete_In.ManReqs2.24,
			In_Manual_SideB_Command:= Discrete_In.ManReqs2.25,
			SideA_Indicator:= FALSE,
			SideB_Indicator:= FALSE,
			TurnOn_SideA_SOL=> N101.Q.24,
			TurnOn_SideB_SOL=> N101.Q.25,
			TurnOn_SideA_Indicator=> Manual_Indicators2.24,
			TurnOn_SideB_Indicator=> Manual_Indicators2.25
			 );
		Valve29FB.In_Auto_SideA_Command:= FALSE;
		Valve29FB.In_Auto_SideB_Command:= FALSE;


	(*Valve 30, A+B*)
	(*spare*)
		Valve30FB
			(
			Enable_Motion:= Enable_Motion ,
			Enable_Latch:= TRUE,					(*Enabling Runs Valve as detent type (maintained solenoids*)
			Enable_SideA_PreCharge:= FALSE,		(*Enabling Turns Side A PreCharge Active, reset when Side B is energized in Auto*)
			Enable_SideB_PreCharge:= FALSE,		(*Enabling Turns Side B PreCharge Active, reset when Side A is energized in Auto*)
			PreCharge_Time:= T#0.10S,
			Enable_Auto_Commands:= In_Auto,
			Enable_Manual_Commands:= In_Manual AND All_Robots_Clear,
			In_Manual_SideA_Command:= Discrete_In.ManReqs2.26,
			In_Manual_SideB_Command:= Discrete_In.ManReqs2.27,
			SideA_Indicator:= FALSE,
			SideB_Indicator:= FALSE,
			TurnOn_SideA_SOL=> N101.Q.26,
			TurnOn_SideB_SOL=> N101.Q.27,
			TurnOn_SideA_Indicator=> Manual_Indicators2.26,
			TurnOn_SideB_Indicator=> Manual_Indicators2.27
			 );
		Valve30FB.In_Auto_SideA_Command:= FALSE;
		Valve30FB.In_Auto_SideB_Command:= FALSE;


	(*Valve 31, A+B*)
	(*spare*)
		Valve31FB
			(
			Enable_Motion:= Enable_Motion ,
			Enable_Latch:= TRUE,					(*Enabling Runs Valve as detent type (maintained solenoids*)
			Enable_SideA_PreCharge:= FALSE,		(*Enabling Turns Side A PreCharge Active, reset when Side B is energized in Auto*)
			Enable_SideB_PreCharge:= FALSE,		(*Enabling Turns Side B PreCharge Active, reset when Side A is energized in Auto*)
			PreCharge_Time:= T#0.10S,
			Enable_Auto_Commands:= In_Auto,
			Enable_Manual_Commands:= In_Manual AND All_Robots_Clear,
			In_Manual_SideA_Command:= Discrete_In.ManReqs2.28,
			In_Manual_SideB_Command:= Discrete_In.ManReqs2.29,
			SideA_Indicator:= FALSE,
			SideB_Indicator:= FALSE,
			TurnOn_SideA_SOL=> N101.Q.28,
			TurnOn_SideB_SOL=> N101.Q.29,
			TurnOn_SideA_Indicator=> Manual_Indicators2.28,
			TurnOn_SideB_Indicator=> Manual_Indicators2.29
			 );
		Valve31FB.In_Auto_SideA_Command:= FALSE;
		Valve31FB.In_Auto_SideB_Command:= FALSE;


	(*Valve 32, A+B*)
	(*spare*)
		Valve32FB
			(
			Enable_Motion:= Enable_Motion ,
			Enable_Latch:= TRUE,					(*Enabling Runs Valve as detent type (maintained solenoids*)
			Enable_SideA_PreCharge:= FALSE,		(*Enabling Turns Side A PreCharge Active, reset when Side B is energized in Auto*)
			Enable_SideB_PreCharge:= FALSE,		(*Enabling Turns Side B PreCharge Active, reset when Side A is energized in Auto*)
			PreCharge_Time:= T#0.10S,
			Enable_Auto_Commands:= In_Auto,
			Enable_Manual_Commands:= In_Manual AND All_Robots_Clear,
			In_Manual_SideA_Command:= Discrete_In.ManReqs2.30,
			In_Manual_SideB_Command:= Discrete_In.ManReqs2.31,
			SideA_Indicator:= FALSE,
			SideB_Indicator:= FALSE,
			TurnOn_SideA_SOL=> N101.Q.30,
			TurnOn_SideB_SOL=> N101.Q.31,
			TurnOn_SideA_Indicator=> Manual_Indicators2.30,
			TurnOn_SideB_Indicator=> Manual_Indicators2.31
			 );
		Valve32FB.In_Auto_SideA_Command:= FALSE;
		Valve32FB.In_Auto_SideB_Command:= FALSE;




















(*end*)
END_ACTION

ACTION ValveBank3:


(*+++++++++++THIS AREA IS CUSTOM PER INSTALLATION AND WILL HAVE TO BE MODIFIED PER +++++++++++++*)
(*+++++++++++THIS AREA IS CUSTOM PER INSTALLATION AND WILL HAVE TO BE MODIFIED PER +++++++++++++*)
(*+++++++++++THIS AREA IS CUSTOM PER INSTALLATION AND WILL HAVE TO BE MODIFIED PER +++++++++++++*)

(*+++++++++++VALVE BANK 3 +++++++++++++*)
(*+++++++++++VALVE BANK 3 +++++++++++++*)
(*+++++++++++VALVE BANK 3 +++++++++++++*)


	(*Valve 33, A+B*)
	(*spare*)
		Valve33FB
			(
			Enable_Motion:= Enable_Motion ,
			Enable_Latch:= TRUE,					(*Enabling Runs Valve as detent type (maintained solenoids*)
			Enable_SideA_PreCharge:= FALSE,		(*Enabling Turns Side A PreCharge Active, reset when Side B is energized in Auto*)
			Enable_SideB_PreCharge:= FALSE,		(*Enabling Turns Side B PreCharge Active, reset when Side A is energized in Auto*)
			PreCharge_Time:= T#0.1S,
			Enable_Auto_Commands:= In_Auto,
			Enable_Manual_Commands:= In_Manual AND All_Robots_Clear,
			In_Manual_SideA_Command:= Discrete_In.ManReqs3.0,
			In_Manual_SideB_Command:= (Discrete_In.ManReqs3.1 OR Discrete_In.Go_Home),
			SideA_Indicator:= FALSE,
			SideB_Indicator:= FALSE,
			TurnOn_SideA_SOL=> N102.Q.0,
			TurnOn_SideB_SOL=> N102.Q.1,
			TurnOn_SideA_Indicator=> Manual_Indicators3.0,
			TurnOn_SideB_Indicator=> Manual_Indicators3.1
			 );
		Valve33FB.In_Auto_SideA_Command:= FALSE;
		Valve33FB.In_Auto_SideB_Command:= FALSE;


	(*Valve 34, A+B*)
	(*spare*)
		Valve34FB
			(
			Enable_Motion:= Enable_Motion ,
			Enable_Latch:= TRUE,					(*Enabling Runs Valve as detent type (maintained solenoids*)
			Enable_SideA_PreCharge:= FALSE,		(*Enabling Turns Side A PreCharge Active, reset when Side B is energized in Auto*)
			Enable_SideB_PreCharge:= FALSE,		(*Enabling Turns Side B PreCharge Active, reset when Side A is energized in Auto*)
			PreCharge_Time:= T#0.10S,
			Enable_Auto_Commands:= In_Auto,
			Enable_Manual_Commands:= In_Manual AND All_Robots_Clear,
			In_Manual_SideA_Command:= Discrete_In.ManReqs3.2,
			In_Manual_SideB_Command:= Discrete_In.ManReqs3.3,
			SideA_Indicator:= FALSE,
			SideB_Indicator:= FALSE,
			TurnOn_SideA_SOL=> N102.Q.2,
			TurnOn_SideB_SOL=> N102.Q.3,
			TurnOn_SideA_Indicator=> Manual_Indicators3.2,
			TurnOn_SideB_Indicator=> Manual_Indicators3.3
			 );
		Valve34FB.In_Auto_SideA_Command:= FALSE;
		Valve34FB.In_Auto_SideB_Command:= FALSE;


	(*Valve 35, A+B*)
	(*spare*)
		Valve35FB
			(
			Enable_Motion:= Enable_Motion ,
			Enable_Latch:= TRUE,					(*Enabling Runs Valve as detent type (maintained solenoids*)
			Enable_SideA_PreCharge:= FALSE,		(*Enabling Turns Side A PreCharge Active, reset when Side B is energized in Auto*)
			Enable_SideB_PreCharge:= FALSE,		(*Enabling Turns Side B PreCharge Active, reset when Side A is energized in Auto*)
			PreCharge_Time:= T#0.10S,
			Enable_Auto_Commands:= In_Auto,
			Enable_Manual_Commands:= In_Manual AND All_Robots_Clear,
			In_Manual_SideA_Command:= Discrete_In.ManReqs3.4,
			In_Manual_SideB_Command:= Discrete_In.ManReqs3.5,
			SideA_Indicator:= FALSE,
			SideB_Indicator:= FALSE,
			TurnOn_SideA_SOL=> N102.Q.4,
			TurnOn_SideB_SOL=> N102.Q.5,
			TurnOn_SideA_Indicator=> Manual_Indicators3.4,
			TurnOn_SideB_Indicator=> Manual_Indicators3.5
			 );
		Valve35FB.In_Auto_SideA_Command:= FALSE;
		Valve35FB.In_Auto_SideB_Command:= FALSE;


	(*Valve 36, A+B*)
	(*spare*)
		Valve36FB
			(
			Enable_Motion:= Enable_Motion ,
			Enable_Latch:= TRUE,					(*Enabling Runs Valve as detent type (maintained solenoids*)
			Enable_SideA_PreCharge:= FALSE,		(*Enabling Turns Side A PreCharge Active, reset when Side B is energized in Auto*)
			Enable_SideB_PreCharge:= FALSE,		(*Enabling Turns Side B PreCharge Active, reset when Side A is energized in Auto*)
			PreCharge_Time:= T#0.10S,
			Enable_Auto_Commands:= In_Auto,
			Enable_Manual_Commands:= In_Manual AND All_Robots_Clear,
			In_Manual_SideA_Command:= Discrete_In.ManReqs3.6,
			In_Manual_SideB_Command:= Discrete_In.ManReqs3.7,
			SideA_Indicator:= FALSE,
			SideB_Indicator:= FALSE,
			TurnOn_SideA_SOL=> N102.Q.6,
			TurnOn_SideB_SOL=> N102.Q.7,
			TurnOn_SideA_Indicator=> Manual_Indicators3.6,
			TurnOn_SideB_Indicator=> Manual_Indicators3.7
			 );
		Valve36FB.In_Auto_SideA_Command:= FALSE;
		Valve36FB.In_Auto_SideB_Command:= FALSE;


	(*Valve 37, A+B*)
	(*spare*)
		Valve37FB
			(
			Enable_Motion:= Enable_Motion ,
			Enable_Latch:= TRUE,					(*Enabling Runs Valve as detent type (maintained solenoids*)
			Enable_SideA_PreCharge:= FALSE,		(*Enabling Turns Side A PreCharge Active, reset when Side B is energized in Auto*)
			Enable_SideB_PreCharge:= FALSE,		(*Enabling Turns Side B PreCharge Active, reset when Side A is energized in Auto*)
			PreCharge_Time:= T#0.10S,
			Enable_Auto_Commands:= In_Auto,
			Enable_Manual_Commands:= In_Manual AND All_Robots_Clear,
			In_Manual_SideA_Command:= Discrete_In.ManReqs3.8,
			In_Manual_SideB_Command:= Discrete_In.ManReqs3.9,
			SideA_Indicator:= FALSE,
			SideB_Indicator:= FALSE,
			TurnOn_SideA_SOL=> N102.Q.8,
			TurnOn_SideB_SOL=> N102.Q.9,
			TurnOn_SideA_Indicator=> Manual_Indicators3.8,
			TurnOn_SideB_Indicator=> Manual_Indicators3.9
			 );
		Valve37FB.In_Auto_SideA_Command:= FALSE;
		Valve37FB.In_Auto_SideB_Command:= FALSE;


	(*Valve 38, A+B*)
	(*spare*)
		Valve38FB
			(
			Enable_Motion:= Enable_Motion ,
			Enable_Latch:= TRUE,					(*Enabling Runs Valve as detent type (maintained solenoids*)
			Enable_SideA_PreCharge:= FALSE,		(*Enabling Turns Side A PreCharge Active, reset when Side B is energized in Auto*)
			Enable_SideB_PreCharge:= FALSE,		(*Enabling Turns Side B PreCharge Active, reset when Side A is energized in Auto*)
			PreCharge_Time:= T#0.10S,
			Enable_Auto_Commands:= In_Auto,
			Enable_Manual_Commands:= In_Manual AND All_Robots_Clear,
			In_Manual_SideA_Command:= Discrete_In.ManReqs3.10,
			In_Manual_SideB_Command:= Discrete_In.ManReqs3.11,
			SideA_Indicator:= FALSE,
			SideB_Indicator:= FALSE,
			TurnOn_SideA_SOL=> N102.Q.10,
			TurnOn_SideB_SOL=> N102.Q.11,
			TurnOn_SideA_Indicator=> Manual_Indicators3.10,
			TurnOn_SideB_Indicator=> Manual_Indicators3.11
			 );
		Valve38FB.In_Auto_SideA_Command:= FALSE;
		Valve38FB.In_Auto_SideB_Command:= FALSE;


	(*Valve 39, A+B*)
	(*spare*)
		Valve39FB
			(
			Enable_Motion:= Enable_Motion ,
			Enable_Latch:= TRUE,					(*Enabling Runs Valve as detent type (maintained solenoids*)
			Enable_SideA_PreCharge:= FALSE,		(*Enabling Turns Side A PreCharge Active, reset when Side B is energized in Auto*)
			Enable_SideB_PreCharge:= FALSE,		(*Enabling Turns Side B PreCharge Active, reset when Side A is energized in Auto*)
			PreCharge_Time:= T#0.10S,
			Enable_Auto_Commands:= In_Auto,
			Enable_Manual_Commands:= In_Manual AND All_Robots_Clear,
			In_Manual_SideA_Command:= Discrete_In.ManReqs3.12,
			In_Manual_SideB_Command:= Discrete_In.ManReqs3.13,
			SideA_Indicator:= FALSE,
			SideB_Indicator:= FALSE,
			TurnOn_SideA_SOL=> N102.Q.12,
			TurnOn_SideB_SOL=> N102.Q.13,
			TurnOn_SideA_Indicator=> Manual_Indicators3.12,
			TurnOn_SideB_Indicator=> Manual_Indicators3.13
			 );
		Valve39FB.In_Auto_SideA_Command:= FALSE;
		Valve39FB.In_Auto_SideB_Command:= FALSE;


	(*Valve 40, A+B*)
	(*spare*)
		Valve40FB
			(
			Enable_Motion:= Enable_Motion ,
			Enable_Latch:= TRUE,					(*Enabling Runs Valve as detent type (maintained solenoids*)
			Enable_SideA_PreCharge:= FALSE,		(*Enabling Turns Side A PreCharge Active, reset when Side B is energized in Auto*)
			Enable_SideB_PreCharge:= FALSE,		(*Enabling Turns Side B PreCharge Active, reset when Side A is energized in Auto*)
			PreCharge_Time:= T#0.10S,
			Enable_Auto_Commands:= In_Auto,
			Enable_Manual_Commands:= In_Manual AND All_Robots_Clear,
			In_Manual_SideA_Command:= Discrete_In.ManReqs3.14,
			In_Manual_SideB_Command:= Discrete_In.ManReqs3.15,
			SideA_Indicator:= FALSE,
			SideB_Indicator:= FALSE,
			TurnOn_SideA_SOL=> N102.Q.14,
			TurnOn_SideB_SOL=> N102.Q.15,
			TurnOn_SideA_Indicator=> Manual_Indicators3.14,
			TurnOn_SideB_Indicator=> Manual_Indicators3.15
			 );
		Valve40FB.In_Auto_SideA_Command:= FALSE;
		Valve40FB.In_Auto_SideB_Command:= FALSE;


	(*Valve 41, A+B*)
	(*spare*)
		Valve41FB
			(
			Enable_Motion:= Enable_Motion ,
			Enable_Latch:= TRUE,					(*Enabling Runs Valve as detent type (maintained solenoids*)
			Enable_SideA_PreCharge:= FALSE,		(*Enabling Turns Side A PreCharge Active, reset when Side B is energized in Auto*)
			Enable_SideB_PreCharge:= FALSE,		(*Enabling Turns Side B PreCharge Active, reset when Side A is energized in Auto*)
			PreCharge_Time:= T#0.10S,
			Enable_Auto_Commands:= In_Auto,
			Enable_Manual_Commands:= In_Manual AND All_Robots_Clear,
			In_Manual_SideA_Command:= Discrete_In.ManReqs3.16,
			In_Manual_SideB_Command:= Discrete_In.ManReqs3.17,
			SideA_Indicator:= FALSE,
			SideB_Indicator:= FALSE,
			TurnOn_SideA_SOL=> N102.Q.16,
			TurnOn_SideB_SOL=> N102.Q.17,
			TurnOn_SideA_Indicator=> Manual_Indicators3.16,
			TurnOn_SideB_Indicator=> Manual_Indicators3.17
			 );
		Valve41FB.In_Auto_SideA_Command:= FALSE;
		Valve41FB.In_Auto_SideB_Command:= FALSE;


	(*Valve 42, A+B*)
	(*spare*)
		Valve42FB
			(
			Enable_Motion:= Enable_Motion ,
			Enable_Latch:= TRUE,					(*Enabling Runs Valve as detent type (maintained solenoids*)
			Enable_SideA_PreCharge:= FALSE,		(*Enabling Turns Side A PreCharge Active, reset when Side B is energized in Auto*)
			Enable_SideB_PreCharge:= FALSE,		(*Enabling Turns Side B PreCharge Active, reset when Side A is energized in Auto*)
			PreCharge_Time:= T#0.10S,
			Enable_Auto_Commands:= In_Auto,
			Enable_Manual_Commands:= In_Manual AND All_Robots_Clear,
			In_Manual_SideA_Command:= Discrete_In.ManReqs3.18,
			In_Manual_SideB_Command:= Discrete_In.ManReqs3.19,
			SideA_Indicator:= FALSE,
			SideB_Indicator:= FALSE,
			TurnOn_SideA_SOL=> N102.Q.18,
			TurnOn_SideB_SOL=> N102.Q.19,
			TurnOn_SideA_Indicator=> Manual_Indicators3.18,
			TurnOn_SideB_Indicator=> Manual_Indicators3.19
			 );
		Valve42FB.In_Auto_SideA_Command:= FALSE;
		Valve42FB.In_Auto_SideB_Command:= FALSE;


	(*Valve 43, A+B*)
	(*spare*)
		Valve43FB
			(
			Enable_Motion:= Enable_Motion ,
			Enable_Latch:= TRUE,					(*Enabling Runs Valve as detent type (maintained solenoids*)
			Enable_SideA_PreCharge:= FALSE,		(*Enabling Turns Side A PreCharge Active, reset when Side B is energized in Auto*)
			Enable_SideB_PreCharge:= FALSE,		(*Enabling Turns Side B PreCharge Active, reset when Side A is energized in Auto*)
			PreCharge_Time:= T#0.10S,
			Enable_Auto_Commands:= In_Auto,
			Enable_Manual_Commands:= In_Manual AND All_Robots_Clear,
			In_Manual_SideA_Command:= Discrete_In.ManReqs3.20,
			In_Manual_SideB_Command:= Discrete_In.ManReqs3.21,
			SideA_Indicator:= FALSE,
			SideB_Indicator:= FALSE,
			TurnOn_SideA_SOL=> N102.Q.20,
			TurnOn_SideB_SOL=> N102.Q.21,
			TurnOn_SideA_Indicator=> Manual_Indicators3.20,
			TurnOn_SideB_Indicator=> Manual_Indicators3.21
			 );
		Valve43FB.In_Auto_SideA_Command:= FALSE;
		Valve43FB.In_Auto_SideB_Command:= FALSE;


	(*Valve 44, A+B*)
	(*spare*)
		Valve44FB
			(
			Enable_Motion:= Enable_Motion ,
			Enable_Latch:= TRUE,					(*Enabling Runs Valve as detent type (maintained solenoids*)
			Enable_SideA_PreCharge:= FALSE,		(*Enabling Turns Side A PreCharge Active, reset when Side B is energized in Auto*)
			Enable_SideB_PreCharge:= FALSE,		(*Enabling Turns Side B PreCharge Active, reset when Side A is energized in Auto*)
			PreCharge_Time:= T#0.10S,
			Enable_Auto_Commands:= In_Auto,
			Enable_Manual_Commands:= In_Manual AND All_Robots_Clear,
			In_Manual_SideA_Command:= Discrete_In.ManReqs3.22,
			In_Manual_SideB_Command:= Discrete_In.ManReqs3.23,
			SideA_Indicator:= FALSE,
			SideB_Indicator:= FALSE,
			TurnOn_SideA_SOL=> N102.Q.22,
			TurnOn_SideB_SOL=> N102.Q.23,
			TurnOn_SideA_Indicator=> Manual_Indicators3.22,
			TurnOn_SideB_Indicator=> Manual_Indicators3.23
			 );
		Valve44FB.In_Auto_SideA_Command:= FALSE;
		Valve44FB.In_Auto_SideB_Command:= FALSE;


	(*Valve 45, A+B*)
	(*spare*)
		Valve45FB
			(
			Enable_Motion:= Enable_Motion ,
			Enable_Latch:= TRUE,					(*Enabling Runs Valve as detent type (maintained solenoids*)
			Enable_SideA_PreCharge:= FALSE,		(*Enabling Turns Side A PreCharge Active, reset when Side B is energized in Auto*)
			Enable_SideB_PreCharge:= FALSE,		(*Enabling Turns Side B PreCharge Active, reset when Side A is energized in Auto*)
			PreCharge_Time:= T#0.10S,
			Enable_Auto_Commands:= In_Auto,
			Enable_Manual_Commands:= In_Manual AND All_Robots_Clear,
			In_Manual_SideA_Command:= Discrete_In.ManReqs3.24,
			In_Manual_SideB_Command:= Discrete_In.ManReqs3.25,
			SideA_Indicator:= FALSE,
			SideB_Indicator:= FALSE,
			TurnOn_SideA_SOL=> N102.Q.24,
			TurnOn_SideB_SOL=> N102.Q.25,
			TurnOn_SideA_Indicator=> Manual_Indicators3.24,
			TurnOn_SideB_Indicator=> Manual_Indicators3.25
			 );
		Valve45FB.In_Auto_SideA_Command:= FALSE;
		Valve45FB.In_Auto_SideB_Command:= FALSE;


	(*Valve 46, A+B*)
	(*spare*)
		Valve46FB
			(
			Enable_Motion:= Enable_Motion ,
			Enable_Latch:= TRUE,					(*Enabling Runs Valve as detent type (maintained solenoids*)
			Enable_SideA_PreCharge:= FALSE,		(*Enabling Turns Side A PreCharge Active, reset when Side B is energized in Auto*)
			Enable_SideB_PreCharge:= FALSE,		(*Enabling Turns Side B PreCharge Active, reset when Side A is energized in Auto*)
			PreCharge_Time:= T#0.10S,
			Enable_Auto_Commands:= In_Auto,
			Enable_Manual_Commands:= In_Manual AND All_Robots_Clear,
			In_Manual_SideA_Command:= Discrete_In.ManReqs3.26,
			In_Manual_SideB_Command:= Discrete_In.ManReqs3.27,
			SideA_Indicator:= FALSE,
			SideB_Indicator:= FALSE,
			TurnOn_SideA_SOL=> N102.Q.26,
			TurnOn_SideB_SOL=> N102.Q.27,
			TurnOn_SideA_Indicator=> Manual_Indicators3.26,
			TurnOn_SideB_Indicator=> Manual_Indicators3.27
			 );
		Valve46FB.In_Auto_SideA_Command:= FALSE;
		Valve46FB.In_Auto_SideB_Command:= FALSE;


	(*Valve 47, A+B*)
	(*spare*)
		Valve47FB
			(
			Enable_Motion:= Enable_Motion ,
			Enable_Latch:= TRUE,					(*Enabling Runs Valve as detent type (maintained solenoids*)
			Enable_SideA_PreCharge:= FALSE,		(*Enabling Turns Side A PreCharge Active, reset when Side B is energized in Auto*)
			Enable_SideB_PreCharge:= FALSE,		(*Enabling Turns Side B PreCharge Active, reset when Side A is energized in Auto*)
			PreCharge_Time:= T#0.10S,
			Enable_Auto_Commands:= In_Auto,
			Enable_Manual_Commands:= In_Manual AND All_Robots_Clear,
			In_Manual_SideA_Command:= Discrete_In.ManReqs3.28,
			In_Manual_SideB_Command:= Discrete_In.ManReqs3.29,
			SideA_Indicator:= FALSE,
			SideB_Indicator:= FALSE,
			TurnOn_SideA_SOL=> N102.Q.28,
			TurnOn_SideB_SOL=> N102.Q.29,
			TurnOn_SideA_Indicator=> Manual_Indicators3.28,
			TurnOn_SideB_Indicator=> Manual_Indicators3.29
			 );
		Valve47FB.In_Auto_SideA_Command:= FALSE;
		Valve47FB.In_Auto_SideB_Command:= FALSE;


	(*Valve 48, A+B*)
	(*spare*)
		Valve48FB
			(
			Enable_Motion:= Enable_Motion ,
			Enable_Latch:= TRUE,					(*Enabling Runs Valve as detent type (maintained solenoids*)
			Enable_SideA_PreCharge:= FALSE,		(*Enabling Turns Side A PreCharge Active, reset when Side B is energized in Auto*)
			Enable_SideB_PreCharge:= FALSE,		(*Enabling Turns Side B PreCharge Active, reset when Side A is energized in Auto*)
			PreCharge_Time:= T#0.10S,
			Enable_Auto_Commands:= In_Auto,
			Enable_Manual_Commands:= In_Manual AND All_Robots_Clear,
			In_Manual_SideA_Command:= Discrete_In.ManReqs3.30,
			In_Manual_SideB_Command:= Discrete_In.ManReqs3.31,
			SideA_Indicator:= FALSE,
			SideB_Indicator:= FALSE,
			TurnOn_SideA_SOL=> N102.Q.30,
			TurnOn_SideB_SOL=> N102.Q.31,
			TurnOn_SideA_Indicator=> Manual_Indicators3.30,
			TurnOn_SideB_Indicator=> Manual_Indicators3.31
			 );
		Valve48FB.In_Auto_SideA_Command:= FALSE;
		Valve48FB.In_Auto_SideB_Command:= FALSE;


























(*end*)
END_ACTION

ACTION Xfer_To_UI:
(*Transfer General Status of Fixture and I/O Images for Display On HMI*)
	Discrete_Image.Status:= Status;
	Discrete_Image.CLFaults1:= CLFaults1;
	Discrete_Image.CLFaults2:= CLFaults2;
	Discrete_Image.CLFaults3:= CLFaults3;
	Discrete_Image.CLFaults4:= CLFaults4;
	Discrete_Image.CLFaulted:= CLFaulted;
	Discrete_Image.PPFaults:= PPFaults;
	Discrete_Image.PPFaults1:= PPFaults1;
	Discrete_Image.PPFaults2:= PPFaults2;
	Discrete_Image.PPFaulted:= PPFaulted;
	Discrete_Image.Model_Data:= Model_ID;
	Discrete_Image.ToolID:= Fix_ID;
	Discrete_Image.ProdCount:= Prod_Count_Out;
	Discrete_Image.CycleTime:= Cycle_Time_Out;
	Discrete_Image.PrevCycleTime:= PrevCycle_Time_Out;
	Discrete_Image.LoadTime:= Load_Time_Out;
	Discrete_Image.WeldTime:= Weld_Time_Out;
	Discrete_Image.UnloadTime:= Unload_Time_Out;

	Discrete_Image.InAuto:= In_Auto_Mode;
	Discrete_Image.InManual:= In_Manual_Mode;
	Discrete_Image.ManInds:= Manual_Indicators1;
	Discrete_Image.ManInds2:= Manual_Indicators2;
	Discrete_Image.ManInds3:= Manual_Indicators3;
	Discrete_Image.At_Home:= Tool_At_Home;
	Discrete_Image.Enable_Motion:= Enable_Motion;
	Discrete_Image.All_Sensors_Off:= All_Sensors_Off;
	Discrete_Image.Bypass_ACKS:= Discrete_In.Bypass_REQS;
	Discrete_Image.CustomApplication_ACKS:= Discrete_In.CustomApplication_REQS;
	Discrete_Image.Fixture_Allow_Model_Change:= Fixture_Allow_Model_Change;
	Discrete_Image.NodeLayout:=NodeLayout;
	Discrete_Image.NodeState:=NodeState;
	
	Discrete_Image.Input_Node_Count:= Discrete_In.Input_Node_Count;
	Discrete_Image.VB_Node_Count:= Discrete_In.VB_Node_Count;
	Discrete_Image.Water_Stand_Count:= Discrete_In.Water_Stand_Count;

	IF  (Discrete_Image.Input_Node_Count < 4)
		THEN Discrete_Image.VB_Screen_Position:= 1;
	ELSIF  (Discrete_Image.Input_Node_Count < 7)
		THEN Discrete_Image.VB_Screen_Position:= 2;
	ELSIF  (Discrete_Image.Input_Node_Count < 10)
		THEN Discrete_Image.VB_Screen_Position:= 3;
	ELSIF  (Discrete_Image.Input_Node_Count < 13)
		THEN Discrete_Image.VB_Screen_Position:= 4;
	ELSIF  (Discrete_Image.Input_Node_Count < 16)
		THEN Discrete_Image.VB_Screen_Position:= 5;
	ELSIF  (Discrete_Image.Input_Node_Count < 19)
		THEN Discrete_Image.VB_Screen_Position:= 6;
	ELSIF  (Discrete_Image.Input_Node_Count < 22)
		THEN Discrete_Image.VB_Screen_Position:= 7;
	ELSIF  (Discrete_Image.Input_Node_Count < 26)
		THEN Discrete_Image.VB_Screen_Position:= 8;
	ELSE
			Discrete_Image.VB_Screen_Position:= 9;
	END_IF;

	Discrete_Image.N00:= N00;
	Discrete_Image.N01:= N01;
	Discrete_Image.N02:= N02;
	Discrete_Image.N03:= N03;
	Discrete_Image.N04:= N04;
	Discrete_Image.N05:= N05;
	Discrete_Image.N06:= N06;
	Discrete_Image.N07:= N07;
	Discrete_Image.N08:= N08;
	Discrete_Image.N09:= N09;
	Discrete_Image.N10:= N10;
	Discrete_Image.N11:= N11;
	Discrete_Image.N12:= N12;
	Discrete_Image.N13:= N13;
	Discrete_Image.N14:= N14;
	Discrete_Image.N15:= N15;
	Discrete_Image.N16:= N16;
	Discrete_Image.N17:= N17;
	Discrete_Image.N18:= N18;
	Discrete_Image.N19:= N19;
	Discrete_Image.N20:= N20;
	Discrete_Image.N21:= N21;
	Discrete_Image.N22:= N22;
	Discrete_Image.N100:= N100;
	Discrete_Image.N100_STAT:= N100_STAT;
	Discrete_Image.N101:= N101;
	Discrete_Image.N101_STAT:= N101_STAT;
	Discrete_Image.N102:= N102;
	Discrete_Image.N102_STAT:= N102_STAT;
	
	(*IsEnabled control For UI screen: Default "IsEnabled == True"*)
	Discrete_Image.Enable_FixtureContext_Clamps:= TRUE;
	Discrete_Image.Enable_FixtureContext_QA:= TRUE;
	Discrete_Image.Enable_FixtureContext_Manual:= TRUE;


	Discrete_Image.ECatSlave_Cable_Breaks:= ECatSlave_Cable_Breaks;

	Discrete_Image.Operator_Performance_Pen:= Production_Report.Shift_Report[0].Prod_Performance;
END_ACTION

END_PROGRAM

(* stored: Version 1.1.0.1, ProductVersion 3.1.4024.12
   POU Fix04: Id {c2e3ad37-105a-4928-8187-bf5565685508}, SpecialFunc None
   Action All_Sensors: Id {8f5035db-04e4-421b-95f8-08c087aa864c}
   Action Cylinders: Id {a2486ea7-7d1b-4b98-b251-492b3bfbec98}
   Action Hardware: Id {cbd45b80-fd18-4406-ab98-b2b72dd084d8}
   Action Production: Id {5abdc824-3875-413b-9ade-84c23ff050db}
   Action Proxies: Id {83f92222-2787-4c05-b15f-4666c3c1ec6a}
   Action Robot_Registration: Id {c557385d-79a9-4c5d-8c6d-a4b1c5c6f36b}
   Action Status_and_Faults: Id {75f51e52-10a9-42ee-9a8c-abb3a9f3c69e}
   Action Task_Fix_Model_IDs: Id {a677123a-a311-416f-b517-fce48dc49c4f}
   Action Tool_States: Id {d84aa2f9-2a95-4540-bc21-e5d077acc41b}
   Action Tool_VBSeq_Repos: Id {abe0982b-2314-46af-87ec-ee2671daedfc}
   Action ValveBank1: Id {2f2a4fa2-2671-47ca-a1ff-7263c875afdd}
   Action ValveBank2: Id {a25ad187-96a3-457c-9300-7373f7298ec2}
   Action ValveBank3: Id {bdb42cc3-dbda-4997-b973-dc76bcb87784}
   Action Xfer_To_UI: Id {2155a409-b889-45aa-bd77-e6b35bca9f9e} *)
